# B&R Automation Studio project Y4_V3_1 (part 4)

#### SeamersCyclic.st - Cyclic code
```iecst
(********************************************************************
 * COPYRIGHT --
 ********************************************************************
 * Program: Seamers
 * File: SeamersCyclic.st
 * Author: nicke
 ********************************************************************
 * Implementation of program Seamers
 ********************************************************************)

PROGRAM _CYCLIC

//	Seamers.ESClear := Control.ESClear ;
//	Seamers.ControlIN := Control.Achieved1 ;
//	Seamers.Detension := Sol20DT1.Auto ;
//	Seamers.BeltsPT := PresetSys.Belt ;
//	Seamers.VacPT := PresetSys.Vac ;
//	Seamers.VacsStopPT := PresetSys.VacsStop ;
//	Seamers.PumpPT := PresetSys.Water ;
//	Seamers.Trips[1] := MS1Belt1.Trip ;
//	Seamers.Trips[2] := MS2Belt2.Trip ;
//	Seamers.Trips[4] := MS9Vac1.Trip ;
//	Seamers.Trips[7] := MS3Belt3.Trip ;
//	Seamers.Trips[8] := MS4Belt4.Trip ;
//	Seamers.Trips[10] := MS10Vac2.Trip ;
//	Seamers.Trips[13] := MS5Belt5.Trip ;
//	Seamers.Trips[14] := MS6Belt6.Trip ;
//	Seamers.Trips[16] := MS11Vac3.Trip ;
//	Seamers.Trips[19] := MS7Belt7.Trip ;
//	Seamers.Trips[20] := MS8Belt8.Trip ;
//	Seamers.Trips[22] := MS12Vac4.Trip ;
//	Seamers.Float[1] := S64Float.In ;
//	Seamers.Float[2] := S65Float.In ;
//	Seamers ();
//	MS1Belt1.Auto := Seamers.BeltOUT[1] ;
//	MS2Belt2.Auto := Seamers.BeltOUT[2] ;
//	MS3Belt3.Auto := Seamers.BeltOUT[3] ;
//	MS4Belt4.Auto := Seamers.BeltOUT[4] ;
//	MS5Belt5.Auto := Seamers.BeltOUT[5] ;
//	MS6Belt6.Auto := Seamers.BeltOUT[6] ;
//	MS7Belt7.Auto := Seamers.BeltOUT[7] ;
//	MS8Belt8.Auto := Seamers.BeltOUT[8] ;
//	MS9Vac1.Auto := Seamers.VacOUT[1] ;
//	MS11Vac3.Auto := Seamers.VacOUT[2] ;
//	MS10Vac2.Auto := Seamers.VacOUT[3] ;
//	MS12Vac4.Auto := Seamers.VacOUT[4] ;
//	Sol19Pump.Auto := Seamers.PumpOUT[0] ;
//	MS13Water1.Auto := Seamers.PumpOUT[1] ;
//	MS14Water2.Auto := Seamers.PumpOUT[2] ;
//	Seamers.StartAllDisp ;

	(*
	Intercept Interval delay TO be cumulative value OF time that spray nozzles are on (when seaming)
	Use counter FOR scans instead OF TON delay.
	CASE statement OF count FOR interval. Keep TON FOR Open delay.

	Timer in system, as glass is coming round, and times out, pauses line, shuts off the water pump AND vacuum pump FOR a few seconds FOR the bladder TO drain.
	Interval delay between drains.
	*)
	SeamersII.Control.Achieved := Control.Achieved1;
	SeamersII.Control.ESClear := Control.ESClear;
	SeamersII.Detension := Sol20DT1.Auto;
	SeamersII.PresetSys.Belt := PresetSys.Belt;
	SeamersII.PresetSys.Vac := PresetSys.Vac;
	SeamersII.PresetSys.VacsStop := PresetSys.VacsStop;
	SeamersII.PresetSys.Water := PresetSys.Water;
	SeamersII.Trips := SysTemp.Alarms;
	SeamersII.Float[1] := S64Float.In;
	SeamersII.SeekBlock[1] := Ax1.Block;
	SeamersII.SeekBlock[2] := Ax2.Block;
	SeamersII.InterceptInterval := InterceptPT.IntervalPT;
	SeamersII.InterceptOpen := InterceptPT.OpenPT;
	SeamersII ();
	MS1Belt1.Auto := SeamersII.BeltOUT[1];
	MS2Belt2.Auto := SeamersII.BeltOUT[2];
	MS3Belt3.Auto := SeamersII.BeltOUT[3];
	MS4Belt4.Auto := SeamersII.BeltOUT[4];
	MS5Belt5.Auto := SeamersII.BeltOUT[5];
	MS6Belt6.Auto := SeamersII.BeltOUT[6];
	MS7Belt7.Auto := SeamersII.BeltOUT[7];
	MS8Belt8.Auto := SeamersII.BeltOUT[8];
	MS9Vac1.Auto := SeamersII.VacOUT[1];
	MS10Vac2.Auto := SeamersII.VacOUT[2];
	MS11Vac3.Auto := SeamersII.VacOUT[3];
	MS12Vac4.Auto := SeamersII.VacOUT[4];
	Sol19Pump.Auto := SeamersII.ValveOUT[2];
	MS13Water1.Auto := SeamersII.PumpOUT[1];

	// NEW SPRAY NOZZLE CONTROL BASED ON U21
	// TURN ON SECOND PUMP WHEN FIRST VACUUM PUMP IS ON
	MS14Water2.Auto := (MS9Vac1.Auto) OR(MS11Vac3.Auto);
	IF(SeamersII.TransportMode)THEN
		MS14Water2.Auto := FALSE;
	END_IF
	IF NOT(S65Float.In)THEN
		MS14Water2.Auto := FALSE;
	END_IF

	// DON'T USE PRE TRACKING. TURNS SPRAY OFF
//	Spray1.PreTracking := 0; //CHANGE IF PRETRACKING REQUIRED
	Spray1.Track[0] := Track004.Active;
	Spray1.Track[1] := Track005.Active AND NOT(Tracking00.Blocked);
	Spray1.Track[2] := Track101.Active;
	Spray1.Track[3] := Track104.Active;
	Spray1.VacuumStopDelay := PresetSys.VacsStop;
	Spray1.NozzlePerm := NozzlePerm;
	Spray1.Vacuum := MS10Vac2.Auto;
	Spray1.AutoStart := SeamersII.AutoStart[1];
	Spray1.Control := Control.Achieved1;
	Spray1.TransportMode := SeamersII.TransportMode;
	Spray1 ();
	Sol37Spray.Auto := Spray1.Spray;// UNCOMMENT AFTER TESTING

	//ADD CONDITIONS TO RESET SEQUENCE FROM ALL CASES.

	// DON'T USE PRE TRACKING. TURNS SPRAY OFF
	Spray2.Track[0] := Track114.Active;
	Spray2.Track[1] := Track115.Active AND NOT(Tracking11.Blocked);
	Spray2.Track[2] := Track201.Active;
	Spray2.Track[3] := Track204.Active;
	Spray2.VacuumStopDelay := PresetSys.VacsStop;
	Spray2.NozzlePerm := NozzlePerm;
	Spray2.Vacuum := MS10Vac2.Auto;
	Spray2.AutoStart := SeamersII.AutoStart[1];
	Spray2.Control := Control.Achieved1;
	Spray2.TransportMode := SeamersII.TransportMode;
	Spray2 ();
	Sol47Spray.Auto := Spray2.Spray; //UNCOMMENT AFTER TESTING

	//RECIRCULATION VALVE - OPERATE WHEN BOTH SPRAY NOZZLE SOLENOIDS ARE OFF
	Sol53Recirc.Auto := FALSE;
	IF(Spray1.Nozzle.Seq >= NC_CleanDone) AND(Spray2.Nozzle.Seq >= NC_CleanDone)THEN
		IF(Sol37Spray.Auto = FALSE) AND(Sol47Spray.Auto = FALSE)THEN
			Sol53Recirc.Auto := TRUE;
		END_IF
	END_IF

END_PROGRAM
```

### Program Logical/System/SensorInput (IEC) - Anti blip for sensor inputs

#### SensorInputCyclic.st - Cyclic code
```iecst
//*******************************************************************
// * COPYRIGHT --
// ********************************************************************
// * Program: SensorInput
// * File: SensorInputCyclic.st
// * Author: nicke
// ********************************************************************
// * Implementation of program SensorInput
// *******************************************************************//

PROGRAM _CYCLIC

	Speeds.SpeedBatch:= LIMIT(1, Speeds.SpeedBatch, 60);
	Speeds.SpeedCntr:= LIMIT(1, Speeds.SpeedCntr, 60);
	Speeds.SpeedEntry:= LIMIT(1, Speeds.SpeedEntry, 60);
	Speeds.SpeedExit:= LIMIT(1, Speeds.SpeedExit, 60);
	Speeds.SpeedLaser:= LIMIT(1, Speeds.SpeedLaser, 60);
	Speeds.SpeedMax:= LIMIT(1, Speeds.SpeedMax, 60);
	Speeds.SpeedSeam:= LIMIT(1, Speeds.SpeedSeam, 60);
	Speeds.SpeedSlow:= LIMIT(1, Speeds.SpeedSlow, 60);
	Speeds.SpeedTrans:= LIMIT(1, Speeds.SpeedTrans, 60);
	Speeds.SpeedWash:= LIMIT(1, Speeds.SpeedWash, 60);
	Speeds.SpeedSeamSlow:= LIMIT(1, Speeds.SpeedSeamSlow, 60);

	//FILTER SENSOR 1 INPUT TO ELIMINATE FALSE READINGS
	//FB INPUTS
	Sensor1.SensorIN := S1Photo.In ;
	Sensor1.SpeedON := Speeds.SpeedTrans ;
	Sensor1.SpeedOFF := Speeds.SpeedSeam ;
	//CALL FB
	Sensor1 ();
	//FB OUTPUT
	S1Photo.Int := Sensor1.SensorOUT ;

	//FILTER SENSOR 2 INPUT TO ELIMINATE FALSE READINGS
	//FB INPUTS
	Sensor2.SensorIN := S2Photo.In ;
	Sensor2.SpeedON := Speeds.SpeedSlow ;
	Sensor2.SpeedOFF := Speeds.SpeedSeam ;
	//CALL FB
	Sensor2 ();
	//FB OUTPUT
	S2Photo.Int := Sensor2.SensorOUT ;

	//FILTER SENSOR 3 INPUT TO ELIMINATE FALSE READINGS
	//FB INPUTS
	Sensor3.SensorIN := S3Photo.In ;
	Sensor3.SpeedON := Speeds.SpeedSeam ;
	Sensor3.SpeedOFF := Speeds.SpeedSeam ;
	//CALL FB
	Sensor3 ();
	//FB OUTPUT
	S3Photo.Int := Sensor3.SensorOUT ;

	//FILTER SENSOR 4 INPUT TO ELIMINATE FALSE READINGS
	//FB INPUTS
	Sensor4.SensorIN := S4Photo.In ;
	Sensor4.SpeedON := Speeds.SpeedSeam ;
	Sensor4.SpeedOFF := Speeds.SpeedSeam ;
	//CALL FB
	Sensor4 ();
	//FB OUTPUT
	S4Photo.Int := Sensor4.SensorOUT ;

	//FILTER SENSOR 5 INPUT TO ELIMINATE FALSE READINGS
	//FB INPUTS
	Sensor5.SensorIN := S5Photo.In ;
	Sensor5.SpeedON := Speeds.SpeedTrans ;
	Sensor5.SpeedOFF := Speeds.SpeedSeam ;
	//CALL FB
	Sensor5 ();
	//FB OUTPUT
	S5Photo.Int := Sensor5.SensorOUT ;

	//FILTER SENSOR 6 INPUT TO ELIMINATE FALSE READINGS
	//FB INPUTS
	Sensor6.SensorIN := S6Photo.In ;
	Sensor6.SpeedON := Speeds.SpeedSlow ;
	Sensor6.SpeedOFF := Speeds.SpeedSeam ;
	//CALL FB
	Sensor6 ();
	//FB OUTPUT
	S6Photo.Int := Sensor6.SensorOUT ;

	//FILTER SENSOR 7 INPUT TO ELIMINATE FALSE READINGS
	//FB INPUTS
	Sensor7.SensorIN := S7Photo.In ;
	Sensor7.SpeedON := Speeds.SpeedSeam ;
	Sensor7.SpeedOFF := Speeds.SpeedSeam ;
	//CALL FB
	Sensor7 ();
	//FB OUTPUT
	S7Photo.Int := Sensor7.SensorOUT ;

	//FILTER SENSOR 8 INPUT TO ELIMINATE FALSE READINGS
	//FB INPUTS
	Sensor8.SensorIN := S8Photo.In ;
	Sensor8.SpeedON := Speeds.SpeedSeam ;
	Sensor8.SpeedOFF := Speeds.SpeedSeam ;
	//CALL FB
	Sensor8 ();
	//FB OUTPUT
	S8Photo.Int := Sensor8.SensorOUT ;

	//FILTER SENSOR 9 INPUT TO ELIMINATE FALSE READINGS
	//FB INPUTS
	Sensor9.SensorIN := S9Photo.In ;
	Sensor9.SpeedON := Speeds.SpeedSeam ;
	Sensor9.SpeedOFF := Speeds.SpeedSeam ;
	//CALL FB
	Sensor9 ();
	//FB OUTPUT
	S9Photo.Int := Sensor9.SensorOUT ;

	//FILTER SENSOR 12 INPUT TO ELIMINATE FALSE READINGS
	//FB INPUTS
	Sensor12.SensorIN := S12Photo.In ;
	Sensor12.SpeedON := Speeds.SpeedSeam ;
	Sensor12.SpeedOFF := Speeds.SpeedTrans ;
	//CALL FB
	Sensor12 ();
	//FB OUTPUT
	S12Photo.Int := Sensor12.SensorOUT ;

	//FILTER SENSOR 13 INPUT TO ELIMINATE FALSE READINGS
	//FB INPUTS
	Sensor13.SensorIN := S13Photo.In ;
	Sensor13.SpeedON := Speeds.SpeedExit ;
	Sensor13.SpeedOFF := Speeds.SpeedExit ;
	//CALL FB
	Sensor13 ();
	//FB OUTPUT
	S13Photo.Int := Sensor13.SensorOUT ;

	//FILTER SENSOR 14 INPUT TO ELIMINATE FALSE READINGS
	//FB INPUTS
	Sensor14.SensorIN := S14Photo.In ;
	Sensor14.SpeedON := Speeds.SpeedExit ;
	Sensor14.SpeedOFF := Speeds.SpeedExit ;
	//CALL FB
	Sensor14 ();
	//FB OUTPUT
	S14Photo.Int := Sensor14.SensorOUT ;

	//FILTER SENSOR 15 INPUT TO ELIMINATE FALSE READINGS
	//FB INPUTS
	Sensor15.SensorIN := S15Photo.In ;
	Sensor15.SpeedON := Speeds.SpeedExit ;
	Sensor15.SpeedOFF := Speeds.SpeedExit ;
	//CALL FB
	Sensor15 ();
	//FB OUTPUT
	S15Photo.Int := Sensor15.SensorOUT ;

	//FILTER SENSOR 16 INPUT TO ELIMINATE FALSE READINGS
	//FB INPUTS
	Sensor16.SensorIN := S16Photo.In ;
	Sensor16.SpeedON := Speeds.SpeedExit ;
	Sensor16.SpeedOFF := Speeds.SpeedExit ;
	//CALL FB
	Sensor16 ();
	//FB OUTPUT
	S16Photo.Int := Sensor16.SensorOUT ;

	//FILTER SENSOR 17 INPUT TO ELIMINATE FALSE READINGS
	//FB INPUTS
	Sensor17.SensorIN := S17Photo.In ;
	Sensor17.SpeedON := Speeds.SpeedExit ;
	Sensor17.SpeedOFF := Speeds.SpeedExit ;
	//CALL FB
	Sensor17 ();
	//FB OUTPUT
	S17Photo.Int := Sensor17.SensorOUT ;

	//FILTER SENSOR 18 INPUT TO ELIMINATE FALSE READINGS
	//FB INPUTS
	Sensor18.SensorIN := S18Photo.In ;
	Sensor18.SpeedON := Speeds.SpeedCntr ;
	Sensor18.SpeedOFF := Speeds.SpeedCntr ;
	//CALL FB
	Sensor18 ();
	//FB OUTPUT
	S18Photo.Int := Sensor18.SensorOUT ;

	//FILTER SENSOR 19 INPUT TO ELIMINATE FALSE READINGS
	//FB INPUTS
	Sensor19.SensorIN := S19Photo.In ;
	Sensor19.SpeedON := Speeds.SpeedBatch ;
	Sensor19.SpeedOFF := Speeds.SpeedBatch ;
	//CALL FB
	Sensor19 ();
	//FB OUTPUT
	S19Photo.Int := Sensor19.SensorOUT ;

	//FILTER SENSOR 20 INPUT TO ELIMINATE FALSE READINGS
	//FB INPUTS
	Sensor20.SensorIN := S20Photo.In ;
	Sensor20.SpeedON := Speeds.SpeedBatch ;
	Sensor20.SpeedOFF := Speeds.SpeedBatch ;
	//CALL FB
	Sensor20 ();
	//FB OUTPUT
	S20Photo.Int := Sensor20.SensorOUT ;

	//FILTER SENSOR 21 INPUT TO ELIMINATE FALSE READINGS
	//FB INPUTS
	Sensor21.SensorIN := S21Photo.In ;
	Sensor21.SpeedON := Speeds.SpeedBatch ;
	Sensor21.SpeedOFF := Speeds.SpeedWash ;
	//CALL FB
	Sensor21 ();
	//FB OUTPUT
	S21Photo.Int := Sensor21.SensorOUT ;

END_PROGRAM
```

### Program Logical/System/Process (IEC) - Operation information

#### ProcessCyclic.st - Cyclic code
```iecst
(********************************************************************
 * COPYRIGHT -ASHTON INDUSTRIAL 2016-
 ********************************************************************
 * Program: Process
 * Author: NE
 ********************************************************************)

PROGRAM _CYCLIC

	//CALCULATION FOR MACHINE RUN TIME. DISPLAYED IN YY:DD:HH:MM
	//FB INPUTS
	RunTime1.On := Control.Achieved1 ;
	RunTime1.TotReset := Reset.Total ;
	RunTime1.ShftReset := Reset.Time ;
	RunTime1.TotMinIn := Data.TotalMins ;
	RunTime1.TotHrIn := Data.TotalHrs ;
	RunTime1.TotDayIn := Data.TotalDays ;
	RunTime1.TotYrIn := Data.TotalYrs ;
	RunTime1.ShftMinIn := Data.ShiftMins ;
	RunTime1.ShftHrIn := Data.ShiftHrs ;
	RunTime1.ShftDayIn := Data.ShiftDays ;
	RunTime1.ShftYrIn := Data.ShiftYrs ;
	//CALL FB
	RunTime1();
	//FB OUTPUTS
	Data.TotalMins := RunTime1.TotMin ;
	Data.TotalHrs := RunTime1.TotHr ;
	Data.TotalDays := RunTime1.TotDay ;
	Data.TotalYrs := RunTime1.TotYr ;
	Data.ShiftMins := RunTime1.ShftMin ;
	Data.ShiftHrs := RunTime1.ShftHr ;
	Data.ShiftDays := RunTime1.ShftDay ;
	Data.ShiftYrs := RunTime1.ShftYr ;

	//CALCULATE BELT GRIND TIMES FOR WIDTH. DISPLAYED IN DD:HH:MM:SS
	//TRACKING BIT TRIGGER FOR CALCULATION
	GrindFB1.On := FALSE ;
	GrindFB1M.On := FALSE ;
	IF EDGEPOS(Seaming.Stop2) THEN
		GrindFB1.On := TRUE ;
		GrindFB1M.On := TRUE ;
	END_IF

	//FB INPUTS
	GrindFB1.TotReset := Reset.Total ;
	GrindFB1.ShftReset := Reset.Grind ;
	GrindFB1M.ShftReset := MeterageReset1.Reset ;
	IF (ProcessMode.In) THEN
		GrindFB1.Speed := Speeds.SpeedSeamSlow;
	ELSE
		GrindFB1.Speed := Speeds.SpeedSeam ;
	END_IF
	GrindFB1.Measured := Ax2.Measure/10 ;
	GrindFB1.TotMSIn := Grind1.TotalMs ;
	GrindFB1.TotSecIn := Grind1.TotalSec ;
	GrindFB1.TotMinIn := Grind1.TotalMin ;
	GrindFB1.TotHrIn := Grind1.TotalHr ;
	GrindFB1.TotDayIn := Grind1.TotalDay ;
	GrindFB1.ShftMSIn := Grind1.ShiftMs ;
	GrindFB1.ShftSecIn := Grind1.ShiftSec ;
	GrindFB1.ShftMinIn := Grind1.ShiftMin ;
	GrindFB1.ShftHrIn := Grind1.ShiftHr ;
	GrindFB1.ShftDayIn := Grind1.ShiftDay ;
	GrindFB1.TotMtrs1In := Grind1.TotalMLow ;
	GrindFB1.TotMtrs2In := Grind1.TotalMUpp ;
	GrindFB1.TotFt1In := Grind1.TotalFtLow ;
	GrindFB1.TotFt2In := Grind1.TotalFtUpp ;
	GrindFB1M.Measured := GrindFB1.Measured;
 	GrindFB1M.ShftMtrs1In := Grind1.ShiftMLow ;
	GrindFB1M.ShftMtrs2In := Grind1.ShiftMUpp ;
	GrindFB1.ShftFt1In := Grind1.ShiftFtLow ;
	GrindFB1.ShftFt2In := Grind1.ShiftFtUpp ;
	//CALL FB
	GrindFB1();
	GrindFB1M ();
	//FB OUTPUTS
	Grind1.TotalMs := GrindFB1.TotMS ;
	Grind1.TotalSec := GrindFB1.TotSec ;
	Grind1.TotalMin := GrindFB1.TotMin ;
	Grind1.TotalHr := GrindFB1.TotHr ;
	Grind1.TotalDay := GrindFB1.TotDay ;
	Grind1.ShiftMs := GrindFB1.ShftMS ;
	Grind1.ShiftSec := GrindFB1.ShftSec ;
	Grind1.ShiftMin := GrindFB1.ShftMin ;
	Grind1.ShiftHr := GrindFB1.ShftHr ;
	Grind1.ShiftDay := GrindFB1.ShftDay ;
	Grind1.TotalMLow := GrindFB1.TotMtrs1 ;
	Grind1.TotalMUpp := GrindFB1.TotMtrs2 ;
	Grind1.TotalFtLow := GrindFB1.TotFt1 ;
	Grind1.TotalFtUpp := GrindFB1.TotFt2 ;
	Grind1.ShiftMLow := GrindFB1M.ShftMtrs1 ;
	Grind1.ShiftMUpp := GrindFB1M.ShftMtrs2 ;
	Grind1.ShiftFtLow := GrindFB1.ShftFt1 ;
	Grind1.ShiftFtUpp := GrindFB1.ShftFt2 ;

	//CALCULATE BELT GRIND TIMES FOR LENGTH. DISPLAYED IN DD:HH:MM:SS
	//TRACKING BIT TRIGGER FOR CALCULATION
	GrindFB2.On := FALSE ;
	GrindFB2M.On := FALSE ;
	IF EDGEPOS(Seaming.Stop2) THEN
		GrindFB2.On := TRUE ;
		GrindFB2M.On := TRUE ;
	END_IF
	//FB INPUTS
	GrindFB2.TotReset := Reset.Total ;
	GrindFB2.ShftReset := Reset.Grind ;
	GrindFB2M.ShftReset := MeterageReset2.Reset ;
	IF (ProcessMode.In) THEN
		GrindFB2.Speed := Speeds.SpeedSeamSlow;
	ELSE
		GrindFB2.Speed := Speeds.SpeedSeam ;
	END_IF
	GrindFB2.Measured := Tracking20.Length ;
	GrindFB2.TotMSIn := Grind2.TotalMs ;
	GrindFB2.TotSecIn := Grind2.TotalSec ;
	GrindFB2.TotMinIn := Grind2.TotalMin ;
	GrindFB2.TotHrIn := Grind2.TotalHr ;
	GrindFB2.TotDayIn := Grind2.TotalDay ;
	GrindFB2.ShftMSIn := Grind2.ShiftMs ;
	GrindFB2.ShftSecIn := Grind2.ShiftSec ;
	GrindFB2.ShftMinIn := Grind2.ShiftMin ;
	GrindFB2.ShftHrIn := Grind2.ShiftHr ;
	GrindFB2.ShftDayIn := Grind2.ShiftDay ;
	GrindFB2.TotMtrs1In := Grind2.TotalMLow ;
	GrindFB2.TotMtrs2In := Grind2.TotalMUpp ;
	GrindFB2.TotFt1In := Grind2.TotalFtLow ;
	GrindFB2.TotFt2In := Grind2.TotalFtUpp ;
	GrindFB2M.Measured := GrindFB2.Measured;
	GrindFB2M.ShftMtrs1In := Grind2.ShiftMLow ;
	GrindFB2M.ShftMtrs2In := Grind2.ShiftMUpp ;
	GrindFB2.ShftFt1In := Grind2.ShiftFtLow ;
	GrindFB2.ShftFt2In := Grind2.ShiftFtUpp ;
	//CALL FB
	GrindFB2();
	GrindFB2M();
	//FB OUTPUTS
	Grind2.TotalMs := GrindFB2.TotMS ;
	Grind2.TotalSec := GrindFB2.TotSec ;
	Grind2.TotalMin := GrindFB2.TotMin ;
	Grind2.TotalHr := GrindFB2.TotHr ;
	Grind2.TotalDay := GrindFB2.TotDay ;
	Grind2.ShiftMs := GrindFB2.ShftMS ;
	Grind2.ShiftSec := GrindFB2.ShftSec ;
	Grind2.ShiftMin := GrindFB2.ShftMin ;
	Grind2.ShiftHr := GrindFB2.ShftHr ;
	Grind2.ShiftDay := GrindFB2.ShftDay ;
	Grind2.TotalMLow := GrindFB2.TotMtrs1 ;
	Grind2.TotalMUpp := GrindFB2.TotMtrs2 ;
	Grind2.TotalFtLow := GrindFB2.TotFt1 ;
	Grind2.TotalFtUpp := GrindFB2.TotFt2 ;
	Grind2.ShiftMLow := GrindFB2M.ShftMtrs1 ;
	Grind2.ShiftMUpp := GrindFB2M.ShftMtrs2 ;
	Grind2.ShiftFtLow := GrindFB2.ShftFt1 ;
	Grind2.ShiftFtUpp := GrindFB2.ShftFt2 ;

	//COMPARE SHIFT METERS AND SET WARNING WHEN GREATER
	Meterage1 := FB_HIDE;
	Meterage2 := FB_HIDE;
	Warn.Timeout[30] := FALSE;
	Warn.Timeout[31] := FALSE;
	IF (Grind1.ShiftMLow > TrackDelayPT.PTTrack913) THEN
		Meterage1 := FB_SHOW;
		Warn.Timeout[30] := TRUE;
	END_IF
	IF (Grind2.ShiftMLow > TrackDelayPT.PTTrack922) THEN
		Meterage2 := FB_SHOW;
		Warn.Timeout[31] := TRUE;
	END_IF

	//PIECE COUNT
	IF EDGENEG(Seaming.Stop2) AND(Control.Achieved1) THEN
		Data.TotalPiece := Data.TotalPiece + 1 ;
		Data.ShiftPiece := Data.ShiftPiece + 1 ;
	END_IF

	//RESET TOTAL
	IF (Reset.Total) THEN
		Data.TotalPiece := 0 ;
	END_IF

	//RESET SHIFT TOTAL
	IF (Reset.Count) THEN
		Data.ShiftPiece := 0 ;
	END_IF

END_PROGRAM
```

### Program Logical/System/IO (IEC) - IO addressing

#### IOCyclic.st - Cyclic code
```iecst
(********************************************************************
 * COPYRIGHT --
 ********************************************************************
 * Program: IO
 * File: IOCyclic.st
 * Author: nicke
 ********************************************************************
 * Implementation of program IO
 ********************************************************************)

PROGRAM _CYCLIC

	IF NOT(Simulation.On) THEN  //DISABLE WHEN SIMULATION RUNNING
		//MAP X2X ST02 TO VARIABLES
		Control.Start := X2X02.P1 ;
		Control.Stop := X2X02.P2 ;
		Control.EStop1 := X2X02.P3 ;
		X2X02.P4 ;
		MS1Belt1.Trip := X2X02.P5 ;
		MS2Belt2.Trip := X2X02.P6 ;
		MS3Belt3.Trip := X2X02.P7 ;
		MS4Belt4.Trip := X2X02.P8 ;
		MS5Belt5.Trip := X2X02.P9 ;
		MS6Belt6.Trip := X2X02.P10 ;
		MS7Belt7.Trip := X2X02.P11 ;
		MS8Belt8.Trip := X2X02.P12 ;
		//MAP X2X ST03 TO VARIABLES
		MS9Vac1.Trip := X2X03.P1 ;
		MS10Vac2.Trip := X2X03.P2 ;
		MS11Vac3.Trip := X2X03.P3 ;
		MS12Vac4.Trip := X2X03.P4 ;
		MS13Water1.Trip := X2X03.P5 ;
		MS14Water2.Trip := X2X03.P6 ;
		X2X03.P7 ;
		X2X03.P8 ;
		X2X03.P9 ;
		X2X03.P10 ;
		X2X03.P11 ;
		ClearBatch.In := X2X03.P12 ;
		//MAP X2X ST04 TO VARIABLES
		X2X04.P1 := Control.Buzzer ;
		X2X04.P2 := Control.OnLmp1 ;
		X2X04.P3 ;
		X2X04.P4 ;
		X2X04.P5 ;
		X2X04.P6 ;
		X2X04.P7 ;
		X2X04.P8 ;
		X2X04.P9 ;
		X2X04.P10 ;
		X2X04.P11 := SEL(Control.Auto,Sol24DG1B.Test,Sol24DG1B.Auto) ;
		X2X04.P12 := Filstar.Out ;
		//MAP X2X ST08 TO VARIABLES
		X2X08.P1 := SEL(Control.Auto,MS1Belt1.Test,MS1Belt1.Auto) ;
		X2X08.P2 := SEL(Control.Auto,MS2Belt2.Test,MS2Belt2.Auto) ;
		X2X08.P3 := SEL(Control.Auto,MS3Belt3.Test,MS3Belt3.Auto) ;
		X2X08.P4 := SEL(Control.Auto,MS4Belt4.Test,MS4Belt4.Auto) ;
		X2X08.P5 := SEL(Control.Auto,MS5Belt5.Test,MS5Belt5.Auto) ;
		X2X08.P6 := SEL(Control.Auto,MS6Belt6.Test,MS6Belt6.Auto) ;
		X2X08.P7 := SEL(Control.Auto,MS7Belt7.Test,MS7Belt7.Auto) ;
		X2X08.P8 := SEL(Control.Auto,MS8Belt8.Test,MS8Belt8.Auto) ;
		X2X08.P9 := SEL(Control.Auto,MS9Vac1.Test,MS9Vac1.Auto) ;
		X2X08.P10 := SEL(Control.Auto,MS10Vac2.Test,MS10Vac2.Auto) ;
		X2X08.P11 := SEL(Control.Auto,MS11Vac3.Test,MS11Vac3.Auto) ;
		X2X08.P12 := SEL(Control.Auto,MS12Vac4.Test,MS12Vac4.Auto) ;
		X2X08.P13 := SEL(Control.Auto,MS13Water1.Test,MS13Water1.Auto) ;
		X2X08.P14 := SEL(Control.Auto,MS14Water2.Test,MS14Water2.Auto) ;
		X2X08.P15 ;
		X2X08.P16 ;
		//MAP X2X ST10 TO VARIABLES
		S45Foot.In := X2X10.P1 ;
		S1Photo.In := X2X10.P2 ;
		S2Photo.In := X2X10.P3 ;
		S56Lever.In := X2X10.P4 ;
		S30Reed.In := X2X10.P5 ;
		S31Reed.In := X2X10.P6 ;
		LaserBusy.In := X2X10.P7 ;
		X2X10.P8 := LaserFire.Auto ;
		S100Reed.In := X2X10.P9 ;
		X2X10.P10 := SEL(Control.Auto,Sol37Spray.Test,Sol37Spray.Auto) ;
		X2X10.P11 := SEL(Control.Auto,Sol2Blt2.Test,Sol2Blt2.Auto) ;
		X2X10.P12 := SEL(Control.Auto,Sol5Arm1.Test,Sol5Arm1.Auto) ;
		X2X10.P13 := SEL(Control.Auto,Sol6Arm2.Test,Sol6Arm2.Auto) ;
		X2X10.P14 := SEL(Control.Auto,Sol7Arm3.Test,Sol7Arm3.Auto) ;
		X2X10.P15 := SEL(Control.Auto,Sol8Arm4.Test,Sol8Arm4.Auto) ;
		X2X10.P16 := SEL(Control.Auto,Sol20DT1.Test,Sol20DT1.Auto) ;
		//MAP X2X ST11 TO VARIABLES
		S81Photo.In := X2X11.P1 ;
		S82Photo.In := X2X11.P2 ;
		S83Photo.In := X2X11.P3 ;
		S84Photo.In := X2X11.P4 ;
		X2X11.P5 := SEL(Control.Auto,Sol3Blt3.Test,Sol3Blt3.Auto) ;
		X2X11.P6 := SEL(Control.Auto,Sol4Blt4.Test,Sol4Blt4.Auto) ;
		X2X11.P7 := SEL(Control.Auto,Sol21DT2.Test,Sol21DT2.Auto) ;
		S3Photo.In := X2X11.P8 ;
		//MAP X2X ST12 TO VARIABLES
		Servo1POT.In := X2X12.P1 ;
		Servo1NOT.In := X2X12.P2 ;
		S80Origin.In := X2X12.P3 ;
		S101Reed.In := X2X12.P4 ;
		S104Reed.In := X2X12.P5 ;
		S105Reed.In := X2X12.P6 ;
		S106Reed.In := X2X12.P7 ;
		S107Reed.In := X2X12.P8 ;
		S108Reed.In := X2X12.P9 ;
		S109Reed.In := X2X12.P10 ;
		S110Reed.In := X2X12.P11 ;
		S111Reed.In := X2X12.P12 ;
		S112Reed.In := X2X12.P13 ;
		S113Reed.In := X2X12.P14 ;
		S114Reed.In := X2X12.P15 ;
		S115Reed.In := X2X12.P16 ;
		//MAP X2X ST13 TO VARIABLES
		S4Photo.In := X2X13.P1 ;
		S5Photo.In := X2X13.P2 ;
		S6Photo.In := X2X13.P3 ;
		S9Photo.In := X2X13.P4 ;
		S32Reed.In := X2X13.P5 ;
		S33Reed.In := X2X13.P6 ;
		S50Reed.In := X2X13.P7 ;
		S102Reed.In := X2X13.P8 ;
		S103Reed.In := X2X13.P9 ;
		X2X13.P10 := SEL(Control.Auto,Sol30Pal1.Test,Sol30Pal1.Auto) ;
		X2X13.P11 := SEL(Control.Auto,Sol31Pal2.Test,Sol31Pal2.Auto) ;
		X2X13.P12 := SEL(Control.Auto,Sol32Pal3.Test,Sol32Pal3.Auto) ;
		X2X13.P13 := SEL(Control.Auto,Sol33Pal4.Test,Sol33Pal4.Auto) ;
		X2X13.P14 := SEL(Control.Auto,Sol24DG1.Test,Sol24DG1.Auto) ;
		X2X13.P15 := Sol35Laser.Auto ;
		X2X13.P16 := SEL(Control.Auto,Sol19Pump.Test,Sol19Pump.Auto) ;
		//MAP X2X ST14 TO VARIABLES
		X2X14.P1 := SEL(Control.Auto,Sol47Spray.Test,Sol47Spray.Auto) ;
		X2X14.P2 := SEL(Control.Auto,Sol53Recirc.Test,Sol53Recirc.Auto) ;
		X2X14.P3 := SEL(Control.Auto,Sol14Arm6.Test,Sol14Arm6.Auto) ;
		X2X14.P4 := SEL(Control.Auto,Sol15Arm7.Test,Sol15Arm7.Auto) ;
		X2X14.P5 := SEL(Control.Auto,Sol22DT3.Test,Sol22DT3.Auto) ;
		S7Photo.In := X2X14.P6 ;
		S64Float.In := X2X14.P7 ;
		S65Float.In := X2X14.P8 ;
		//MAP X2X ST15 TO VARIABLES
		Servo2POT.In := X2X15.P1 ;
		Servo2NOT.In := X2X15.P2 ;
		S90Origin.In := X2X15.P3 ;
		S12Photo.In := X2X15.P4 ;
		S13Photo.In := X2X15.P5 ;
		S34Reed.In := X2X15.P6 ;
		S35Reed.In := X2X15.P7 ;
		X2X15.P8 ;
		S120Reed.In := X2X15.P9 ;
		S121Reed.In := X2X15.P10 ;
		S122Reed.In := X2X15.P11 ;
		S123Reed.In := X2X15.P12 ;
		S124Reed.In := X2X15.P13 ;
		S125Reed.In := X2X15.P14 ;
		S126Reed.In := X2X15.P15 ;
		S127Reed.In := X2X15.P16 ;
		//MAP X2X ST16 TO VARIABLES
		S91Photo.In := X2X16.P1 ;
		S92Photo.In := X2X16.P2 ;
		S93Photo.In := X2X16.P3 ;
		S94Photo.In := X2X16.P4 ;
		X2X16.P5 := SEL(Control.Auto,Sol12Blt7.Test,Sol12Blt7.Auto) ;
		X2X16.P6 := SEL(Control.Auto,Sol13Blt8.Test,Sol13Blt8.Auto) ;
		X2X16.P7 := SEL(Control.Auto,Sol23DT4.Test,Sol23DT4.Auto) ;
		S8Photo.In := X2X16.P8 ;
		X2X16.P9 := SEL(Control.Auto,Sol40Datum.Test,Sol40Datum.Auto) ;
		X2X16.P10 ;
		X2X16.P11 ;
		X2X16.P12 ;
		S52Reed.In := X2X16.P13 ;
		S53Reed.In := X2X16.P14 ;
		X2X16.P15 ;
		X2X16.P16 ;
		//MAP X2X ST17 TO VARIABLES
		S14Photo.In := X2X17.P1 ;
		S15Photo.In := X2X17.P2 ;
		S16Photo.In := X2X17.P3 ;
		S17Photo.In := X2X17.P4 ;
		S18Photo.In := X2X17.P5 ;
		S36Reed.In := X2X17.P6 ;
		S37Reed.In := X2X17.P7 ;
		S57Lever.In := X2X17.P8 ;
		//MAP X2X ST18 TO VARIABLES
		S19Photo.In := X2X18.P1 ;
		X2X18.P2 ;
		X2X18.P3 ;
		X2X18.P4 ;
		S21Photo.In := X2X18.P5 ;
		X2X18.P6 ;
		S55Lever.In := X2X18.P7 ;
		WashRun.In := X2X18.P8 ;
		FurnReady.In := X2X18.P9 ;
		X2X18.P10 := WashStop.Auto ;
		X2X18.P11 := BatchAtExit.Auto ;
		S48Foot.In := X2X18.P12 ;
		S66PB.In := X2X18.P13 ;
		S58Lever.In := X2X18.P14 ;
		S20Photo.In := X2X18.P15 ;
		X2X18.P16 ; //INPUT CAN BE USED FOR BUTTON OR FOOTPEDAL TO BRING UP NEXT SCREEN ON BATCHING DISPLAY.
		//MAP X2X ST20 TO VARIABLES
		AGVReady.In := X2X20.P1;
		AGVInPosition.In := X2X20.P2;
		AGVReceiving.In := X2X20.P3;
		X2X20.P4;
		X2X20.P5;
		X2X20.P6;
		X2X20.P7;
		X2X20.P8;
		X2X20.P9;
		X2X20.P10;
		AGVAcknowledge.In := X2X20.P11;
		X2X20.P12;
		//MAP X2X ST21 TO VARIABLES
		X2X21.P1 := AGVRequired.Auto;
		X2X21.P2;
		X2X21.P3;
		X2X21.P4;
		X2X21.P5 := AGVReadyToSend.Auto;
		X2X21.P6;
		X2X21.P7 := AGVBatchClear.Auto;
		X2X21.P8 := SizeData.LengthMask;
		X2X21.P9 := SizeData.WidthMask;
		X2X21.P10 := AGVSending.Auto;
		X2X21.P11;
		X2X21.P12;
		//MAP X2X ST22 TO VARIABLES
		X2X22.P1 := SizeData.Sizes[0];
		X2X22.P2 := SizeData.Sizes[1];
		X2X22.P3 := SizeData.Sizes[2];
		X2X22.P4 := SizeData.Sizes[3];
		X2X22.P5 := SizeData.Sizes[4];
		X2X22.P6 := SizeData.Sizes[5];
		X2X22.P7 := SizeData.Sizes[6];
		X2X22.P8 := SizeData.Sizes[7];
		X2X22.P9 := SizeData.Sizes[8];
		X2X22.P10 := SizeData.Sizes[9];
		X2X22.P11 := SizeData.Sizes[10];
		X2X22.P12 := SizeData.Sizes[11];
	END_IF

	//RESET TEST BITS WHEN EXITING TEST SCREENS
	IF NOT(Control.Test) THEN
		Sol24DG1B.Test := FALSE ;
		MS1Belt1.Test := FALSE ;
		MS2Belt2.Test := FALSE ;
		MS3Belt3.Test := FALSE ;
		MS4Belt4.Test := FALSE ;
		MS5Belt5.Test := FALSE ;
		MS6Belt6.Test := FALSE ;
		MS7Belt7.Test := FALSE ;
		MS8Belt8.Test := FALSE ;
		MS9Vac1.Test := FALSE ;
		MS10Vac2.Test := FALSE ;
		MS11Vac3.Test := FALSE ;
		MS12Vac4.Test := FALSE ;
		MS13Water1.Test := FALSE ;
		MS14Water2.Test := FALSE ;
		Sol1Blt1.Test := FALSE ;
		Sol2Blt2.Test := FALSE ;
		Sol5Arm1.Test := FALSE ;
		Sol6Arm2.Test := FALSE ;
		Sol7Arm3.Test := FALSE ;
		Sol8Arm4.Test := FALSE ;
		Sol3Blt3.Test := FALSE ;
		Sol4Blt4.Test := FALSE ;
		Sol19Pump.Test := FALSE ;
		Sol21DT2.Test := FALSE ;
		Sol30Pal1.Test := FALSE ;
		Sol31Pal2.Test := FALSE ;
		Sol32Pal3.Test := FALSE ;
		Sol33Pal4.Test := FALSE ;
		Sol24DG1.Test := FALSE ;
		Sol10Blt5.Test := FALSE ;
		Sol11Blt6.Test := FALSE ;
		Sol14Arm6.Test := FALSE ;
		Sol15Arm7.Test := FALSE ;
		Sol12Blt7.Test := FALSE ;
		Sol13Blt8.Test := FALSE ;
		Sol23DT4.Test := FALSE ;
		Sol37Spray.Test := FALSE;
		Sol40Datum.Test := FALSE ;
		Sol47Spray.Test := FALSE;
		Sol53Recirc.Test := FALSE;
		CL1.Inv.Test := 0 ;
		CS1.Inv.Test := 0 ;
		CV1.Inv.Test := 0 ;
		CC1.Inv.Test := 0 ;
		CC2.Inv.Test := 0 ;
		CS2.Inv.Test := 0 ;
		CV2.Inv.Test := 0 ;
		CC3.Inv.Test := 0 ;
		CC4.Inv.Test := 0 ;
		CB1.Inv.Test := 0 ;
		CB2.Inv.Test := 0 ;
		CRB.Inv.Test := 0 ;
		CRE.Inv.Test := 0 ;
		CLB.Inv.Test := 0 ;
	END_IF

END_PROGRAM
```

### Program Logical/System/Filstar (IEC) - Filstar valve control

#### FilstarCyclic.st - Cyclic code
```iecst
(********************************************************************
 * COPYRIGHT --
 ********************************************************************
 * Program: Filstar
 * File: FilstarCyclic.st
 * Author: nicke
 * Created: February, 2012
 ********************************************************************
 * Implementation of program Filstar
 ********************************************************************)

PROGRAM _INIT

Filstar.Open.IN		:=	TRUE	;

END_PROGRAM

PROGRAM _CYCLIC

(*Delay for filstar valve open*)
Filstar.Open.PT	:=	PresetSys.Filstar[1]	;
Filstar.Open ();
(*Filstar valve control*)
Filstar.Out	:=	Filstar.Open.M	;

IF (Filstar.Open.Q) THEN
	Filstar.Open.IN		:=	FALSE	;
	Filstar.Interval.IN	:=	TRUE	;
END_IF
(*Delay for inteval between valve open*)
Filstar.Interval.PT	:=	PresetSys.Filstar[2]	;
Filstar.Interval ();

IF (Filstar.Interval.Q) THEN
	Filstar.Interval.IN	:= 	FALSE	;
	Filstar.Open.IN		:=	TRUE	;
END_IF

END_PROGRAM
```

### Program Logical/System/LineConfig (IEC) - IO Line Configuration

#### LineConfigCyclic.st - Cyclic code
```iecst
(********************************************************************
 * COPYRIGHT --
 ********************************************************************
 * Program: LineConfig
 * File: LineConfigCyclic.st
 * Author: nicke
 ********************************************************************)
PROGRAM _CYCLIC

	Perms.FLIPARMS1 := 4 ;
	Perms.FLIPARMS2 := 2 ;

	Perms.VersionText	:=	'S/W Version 3.1 02/26'	;

	// DeviceName used for mapping IO to ACOPOS
	Ax1.Node	:=	'SL1.IF1.ST1.IF1.ST12'	;	// Alter to suit each job
	Ax2.Node	:=	'SL1.IF1.ST1.IF1.ST15'	;	// Alter to suit each job

// Servo settings
	Ax1P.AbsMax	:=	40000				;	// Max Size of Axis 1
	Ax1P.AbsMin	:=	3000				;	// Min Size of Axis 1
	Ax2P.AbsMax	:=	25000				;	// Max Size of Axis 2
	Ax2P.AbsMin	:=	2000				;	// Min Size of Axis 2

	// Calculated limits for visu input
	Ax1.Max.Upp		:=	(Ax1P.AbsMax + 50)		;	// Maximum upper limit input
	Ax1.Max.Low		:=	(Ax1P.AbsMax/2)			;	// Maximum lower limit input
	Ax1.Max.UppF	:=	(Ax1P.AbsMax - 2000)	;	// Maximum feed upper limit input
	Ax1.Max.LowF	:=	(Ax1P.AbsMax - 2800)	;	// Maximum feed lower limit input
	Ax1.Max.UppO	:=	(Ax1P.AbsMax + 50)		;	// Maximum origin upper limit input
	Ax1.Max.LowO	:=	(Ax1P.AbsMax - 50)		;	// Maximum origin lower limit input
	Ax1.Min.Upp		:=	(Ax1P.AbsMax/2)			;	// Minimum upper limit input
	Ax1.Min.Low		:=	(Ax1P.AbsMin - 50)		;	// Minimum lower limit input
	Ax1.Min.UppF	:=	(Ax1P.AbsMin + 2000)	;	// Minimum feed upper limit input
	Ax1.Min.LowF	:=	(Ax1P.AbsMin + 3500)	;	// Minimum feed lower limit input
	Ax2.Max.Upp		:=	(Ax2P.AbsMax + 50)		;	// Maximum upper limit input
	Ax2.Max.Low		:=	(Ax2P.AbsMax/2)			;	// Maximum lower limit input
	Ax2.Max.UppF	:=	(Ax2P.AbsMax - 2000)	;	// Maximum feed upper limit input
	Ax2.Max.LowF	:=	(Ax2P.AbsMax - 2800)	;	// Maximum feed lower limit input
	Ax2.Max.UppO	:=	(Ax2P.AbsMax + 50)		;	// Maximum origin upper limit input
	Ax2.Max.LowO	:=	(Ax2P.AbsMax - 50)		;	// Maximum origin lower limit input
	Ax2.Min.Upp		:=	(Ax2P.AbsMax/2)			;	// Minimum upper limit input
	Ax2.Min.Low		:=	(Ax2P.AbsMin - 50)		;	// Minimum lower limit input
	Ax2.Min.UppF	:=	(Ax2P.AbsMin + 2000)	;	// Minimum feed upper limit input
	Ax2.Min.LowF	:=	(Ax2P.AbsMin + 3500)	;	// Minimum feed lower limit input

	//LIMIT INPUT VALUES FOR HMI
	RowPerm.Max		:=	LIMIT(150,RowPerm.Max,2489)	;//98"
	LoadPerm.Max	:=	LIMIT(300,LoadPerm.Max,5004);//197"

END_PROGRAM
```

### Package Logical/Automatic - Automatic sequencing

### Automatic.var - Package variables
```iecst
(********************************************************************
 * COPYRIGHT --
 ********************************************************************
 * Package: Automatic
 * File: Automatic.var
 * Author: nicke
 * Created: February, 2012
 ********************************************************************
 * Variables of package Automatic
 ********************************************************************)
VAR
	Belt1 : TrackProc; (*Belt timing control*)
	Belt2 : TrackProc; (*Belt timing control*)
	Belt3 : TrackProc; (*Belt timing control*)
	Belt4 : TrackProc; (*Belt timing control*)
	Belt5 : TrackProc; (*Belt timing control*)
	Belt6 : TrackProc; (*Belt timing control*)
	Belt7 : TrackProc; (*Belt timing control*)
	Belt8 : TrackProc; (*Belt timing control*)
END_VAR
```

### Program Logical/Automatic/ResetInv (IEC) - Reset Inverters Before scan

#### ResetInv.st - Implementation code
```iecst
(********************************************************************
 * COPYRIGHT --
 ********************************************************************
 * Program: ResetInv
 * File: ResetInv.st
 * Author: nicke
 ********************************************************************
 * Implementation of program ResetInv
 ********************************************************************)

PROGRAM _CYCLIC

    //INVERTER CL1 CONTROLS
    //SCALE DISPLAY VALUES OF M/MIN TO FREQUENCY FOR CONVEYOR SET SPEEDS
	CL1.Inv.Reference1[0].x := 00.0 ;
	CL1.Inv.Reference1[0].y := 00.0 ;
	CL1.Inv.Reference1[1].x := ScalePerm.CL1Scale ; //SPEED OF CONVEYOR AT 50HZ. ALTER AS REQUIRED
	CL1.Inv.Reference1[1].y    := 500.0 ;  //500 = 50HZ

	CASE InvPerms.CL1.Analog OF
		NO_ANALOG:
		VOLTAGE_TYPE_1:
			CL1.SpeedAnalog := ((INT_TO_REAL(CL1.Input.AI1R))/(AnalogPerm.CL1.V1.ActAnalog/AnalogPerm.CL1.V1.ActSpeed)) ;
		CURRENT_TYPE_1:
			CL1.SpeedAnalog := ((INT_TO_REAL(CL1.Input.AI3R))/(AnalogPerm.CL1.C1.ActAnalog/AnalogPerm.CL1.C1.ActSpeed)) ;
		CURRENT_TYPE_2:
			CL1.SpeedAnalog := ((INT_TO_REAL(CL1.Input.AI3R)-1638.4)/(AnalogPerm.CL1.C2.ActAnalog/AnalogPerm.CL1.C2.ActSpeed)) ; //1638.4 IS 4mA SHIFT FOR 4-20mA RANGE
		CL1.Inv.Reference1[1].y := 400.0 ; //REDUCE SCALE REFERENCE BY 20% TO ALLOW FOR 4mA SHIFT
	END_CASE
	CL1.SpeedAnalog := LIMIT(1, CL1.SpeedAnalog, 60) ;

	CL1.Inv.Scale1.NoOfPoints := 2 ;
	CL1.Inv.Scale1.ptr_table := ADR(CL1.Inv.Reference1)    ;

	//RESET INVERTER OUTPUTS BEFORE SCAN
	IF NOT(Control.Test) THEN
		memcpy(ADR(CL1.o),ADR(ClearInv),SIZEOF(ClearInv));
	END_IF

	//INVERTER ENABLE CONTROL
	IF(Control.Achieved1) OR(Control.Test) THEN
		IF(CL1.Input.ETAD_06) THEN
			CL1.Output.CMDD_01 := TRUE ;
			CL1.Output.CMDD_02 := TRUE ;
		END_IF
		IF(CL1.Input.ETAD_04) AND(CL1.Input.ETAD_05) THEN
			CL1.Output.CMDD_00 := TRUE ;
		END_IF
	END_IF

	//INVERTER RESET CONTROL
	IF NOT(Control.Achieved1) AND NOT(Control.Test) THEN
		CL1.Output.CMDD_00 := FALSE ;
		CL1.Output.CMDD_01 := FALSE ;
		CL1.Output.CMDD_02 := FALSE ;
		CL1.Output.CMDD_07 := FALSE ;
	END_IF

	//SET INVERTER FREQUENCY
	CL1.Inv.Scale1();
	CL1.o.SpeedRef := CL1.Inv.Scale1.y ;
	CL1.Output.LFR := REAL_TO_INT(CL1.o.SpeedRef) ;

	//INVERTER CS1 CONTROLS
	//SCALE DISPLAY VALUES OF M/MIN TO FREQUENCY FOR CONVEYOR SET SPEEDS
	CS1.Inv.Reference1[0].x := 00.0 ;
	CS1.Inv.Reference1[0].y := 00.0 ;
	CS1.Inv.Reference1[1].x := ScalePerm.CS1Scale ; //SPEED OF CONVEYOR AT 50HZ. ALTER AS REQUIRED
	CS1.Inv.Reference1[1].y    := 500.0 ;  //500 = 50HZ

	CASE InvPerms.CS1.Analog OF
		NO_ANALOG:
		VOLTAGE_TYPE_1:
			CS1.SpeedAnalog := ((INT_TO_REAL(CS1.Input.AI1R))/(AnalogPerm.CS1.V1.ActAnalog/AnalogPerm.CS1.V1.ActSpeed)) ;
		CURRENT_TYPE_1:
			CS1.SpeedAnalog := ((INT_TO_REAL(CS1.Input.AI3R))/(AnalogPerm.CS1.C1.ActAnalog/AnalogPerm.CS1.C1.ActSpeed)) ;
		CURRENT_TYPE_2:
			CS1.SpeedAnalog := ((INT_TO_REAL(CS1.Input.AI3R)-1638.4)/(AnalogPerm.CS1.C2.ActAnalog/AnalogPerm.CS1.C2.ActSpeed)) ; //1638.4 IS 4mA SHIFT FOR 4-20mA RANGE
		CS1.Inv.Reference1[1].y := 400.0 ; //REDUCE SCALE REFERENCE BY 20% TO ALLOW FOR 4mA SHIFT
	END_CASE
	CS1.SpeedAnalog := LIMIT(1, CS1.SpeedAnalog, 60) ;

	CS1.Inv.Scale1.NoOfPoints := 2 ;
	CS1.Inv.Scale1.ptr_table := ADR(CS1.Inv.Reference1)    ;

	//RESET INVERTER OUTPUTS BEFORE SCAN
	IF NOT(Control.Test) THEN
		memcpy(ADR(CS1.o),ADR(ClearInv),SIZEOF(ClearInv));
	END_IF

	//INVERTER ENABLE CONTROL
	IF(Control.Achieved1) OR(Control.Test) THEN
		IF(CS1.Input.ETAD_06) THEN
			CS1.Output.CMDD_01 := TRUE ;
			CS1.Output.CMDD_02 := TRUE ;
		END_IF
		IF(CS1.Input.ETAD_04) AND(CS1.Input.ETAD_05) THEN
			CS1.Output.CMDD_00 := TRUE ;
		END_IF
	END_IF

	//INVERTER RESET CONTROL
	IF NOT(Control.Achieved1) AND NOT(Control.Test) THEN
		CS1.Output.CMDD_00 := FALSE ;
		CS1.Output.CMDD_01 := FALSE ;
		CS1.Output.CMDD_02 := FALSE ;
		CS1.Output.CMDD_07 := FALSE ;
	END_IF

	//SET INVERTER FREQUENCY
	CS1.Inv.Scale1();
	CS1.o.SpeedRef := CS1.Inv.Scale1.y ;
	CS1.Output.LFR := REAL_TO_INT(CS1.o.SpeedRef) ;

	//INVERTER CV1 CONTROLS
	//SCALE DISPLAY VALUES OF M/MIN TO FREQUENCY FOR CONVEYOR SET SPEEDS
	CV1.Inv.Reference1[0].x := 00.0 ;
	CV1.Inv.Reference1[0].y := 00.0 ;
	CV1.Inv.Reference1[1].x := ScalePerm.CV1Scale ; //SPEED OF CONVEYOR AT 50HZ. ALTER AS REQUIRED
	CV1.Inv.Reference1[1].y    := 500.0 ;  //500 = 50HZ

	CASE InvPerms.CV1.Analog OF
		NO_ANALOG:
		VOLTAGE_TYPE_1:
			CV1.SpeedAnalog := ((INT_TO_REAL(CV1.Input.AI1R))/(AnalogPerm.CV1.V1.ActAnalog/AnalogPerm.CV1.V1.ActSpeed)) ;
		CURRENT_TYPE_1:
			CV1.SpeedAnalog := ((INT_TO_REAL(CV1.Input.AI3R))/(AnalogPerm.CV1.C1.ActAnalog/AnalogPerm.CV1.C1.ActSpeed)) ;
		CURRENT_TYPE_2:
			CV1.SpeedAnalog := ((INT_TO_REAL(CV1.Input.AI3R)-1638.4)/(AnalogPerm.CV1.C2.ActAnalog/AnalogPerm.CV1.C2.ActSpeed)) ; //1638.4 IS 4mA SHIFT FOR 4-20mA RANGE
		CV1.Inv.Reference1[1].y := 400.0 ; //REDUCE SCALE REFERENCE BY 20% TO ALLOW FOR 4mA SHIFT
	END_CASE
	CV1.SpeedAnalog := LIMIT(1, CV1.SpeedAnalog, 60) ;

	CV1.Inv.Scale1.NoOfPoints := 2 ;
	CV1.Inv.Scale1.ptr_table := ADR(CV1.Inv.Reference1)    ;

	//RESET INVERTER OUTPUTS BEFORE SCAN
	IF NOT(Control.Test) THEN
		memcpy(ADR(CV1.o),ADR(ClearInv),SIZEOF(ClearInv));
	END_IF

	//INVERTER ENABLE CONTROL
	IF(Control.Achieved1) OR(Control.Test) THEN
		IF(CV1.Input.ETAD_06) THEN
			CV1.Output.CMDD_01 := TRUE ;
			CV1.Output.CMDD_02 := TRUE ;
		END_IF
		IF(CV1.Input.ETAD_04) AND(CV1.Input.ETAD_05) THEN
			CV1.Output.CMDD_00 := TRUE ;
		END_IF
	END_IF

	//INVERTER RESET CONTROL
	IF NOT(Control.Achieved1) AND NOT(Control.Test) THEN
		CV1.Output.CMDD_00 := FALSE ;
		CV1.Output.CMDD_01 := FALSE ;
		CV1.Output.CMDD_02 := FALSE ;
		CV1.Output.CMDD_07 := FALSE ;
	END_IF

	//SET INVERTER FREQUENCY
	CV1.Inv.Scale1();
	CV1.o.SpeedRef := CV1.Inv.Scale1.y ;
	CV1.Output.LFR := REAL_TO_INT(CV1.o.SpeedRef) ;

	//INVERTER CC1 CONTROLS
	//SCALE DISPLAY VALUES OF M/MIN TO FREQUENCY FOR CONVEYOR SET SPEEDS
	CC1.Inv.Reference1[0].x := 00.0 ;
	CC1.Inv.Reference1[0].y := 00.0 ;
	CC1.Inv.Reference1[1].x := ScalePerm.CC1Scale ; //SPEED OF CONVEYOR AT 50HZ. ALTER AS REQUIRED
	CC1.Inv.Reference1[1].y    := 500.0 ;  //500 = 50HZ

	CASE InvPerms.CC1.Analog OF
		NO_ANALOG:
		VOLTAGE_TYPE_1:
			CC1.SpeedAnalog := ((INT_TO_REAL(CC1.Input.AI1R))/(AnalogPerm.CC1.V1.ActAnalog/AnalogPerm.CC1.V1.ActSpeed)) ;
		CURRENT_TYPE_1:
			CC1.SpeedAnalog := ((INT_TO_REAL(CC1.Input.AI3R))/(AnalogPerm.CC1.C1.ActAnalog/AnalogPerm.CC1.C1.ActSpeed)) ;
		CURRENT_TYPE_2:
			CC1.SpeedAnalog := ((INT_TO_REAL(CC1.Input.AI3R)-1638.4)/(AnalogPerm.CC1.C2.ActAnalog/AnalogPerm.CC1.C2.ActSpeed)) ; //1638.4 IS 4mA SHIFT FOR 4-20mA RANGE
		CC1.Inv.Reference1[1].y := 400.0 ; //REDUCE SCALE REFERENCE BY 20% TO ALLOW FOR 4mA SHIFT
	END_CASE
	CC1.SpeedAnalog := LIMIT(1, CC1.SpeedAnalog, 60) ;

	CC1.Inv.Scale1.NoOfPoints := 2 ;
	CC1.Inv.Scale1.ptr_table := ADR(CC1.Inv.Reference1)    ;

	//RESET INVERTER OUTPUTS BEFORE SCAN
	IF NOT(Control.Test) THEN
		memcpy(ADR(CC1.o),ADR(ClearInv),SIZEOF(ClearInv));
	END_IF

	//INVERTER ENABLE CONTROL
	IF(Control.Achieved1) OR(Control.Test) THEN
		IF(CC1.Input.ETAD_06) THEN
			CC1.Output.CMDD_01 := TRUE ;
			CC1.Output.CMDD_02 := TRUE ;
		END_IF
		IF(CC1.Input.ETAD_04) AND(CC1.Input.ETAD_05) THEN
			CC1.Output.CMDD_00 := TRUE ;
		END_IF
	END_IF

	//INVERTER RESET CONTROL
	IF NOT(Control.Achieved1) AND NOT(Control.Test) THEN
		CC1.Output.CMDD_00 := FALSE ;
		CC1.Output.CMDD_01 := FALSE ;
		CC1.Output.CMDD_02 := FALSE ;
		CC1.Output.CMDD_07 := FALSE ;
	END_IF

	//SET INVERTER FREQUENCY
	CC1.Inv.Scale1();
	CC1.o.SpeedRef := CC1.Inv.Scale1.y ;
	CC1.Output.LFR := REAL_TO_INT(CC1.o.SpeedRef) ;

	//INVERTER CC2 CONTROLS
	//SCALE DISPLAY VALUES OF M/MIN TO FREQUENCY FOR CONVEYOR SET SPEEDS
	CC2.Inv.Reference1[0].x := 00.0 ;
	CC2.Inv.Reference1[0].y := 00.0 ;
	CC2.Inv.Reference1[1].x := ScalePerm.CC2Scale ; //SPEED OF CONVEYOR AT 50HZ. ALTER AS REQUIRED
	CC2.Inv.Reference1[1].y    := 500.0 ;  //500 = 50HZ

	CASE InvPerms.CC2.Analog OF
		NO_ANALOG:
		VOLTAGE_TYPE_1:
			CC2.SpeedAnalog := ((INT_TO_REAL(CC2.Input.AI1R))/(AnalogPerm.CC2.V1.ActAnalog/AnalogPerm.CC2.V1.ActSpeed)) ;
		CURRENT_TYPE_1:
			CC2.SpeedAnalog := ((INT_TO_REAL(CC2.Input.AI3R))/(AnalogPerm.CC2.C1.ActAnalog/AnalogPerm.CC2.C1.ActSpeed)) ;
		CURRENT_TYPE_2:
			CC2.SpeedAnalog := ((INT_TO_REAL(CC2.Input.AI3R)-1638.4)/(AnalogPerm.CC2.C2.ActAnalog/AnalogPerm.CC2.C2.ActSpeed)) ; //1638.4 IS 4mA SHIFT FOR 4-20mA RANGE
		CC2.Inv.Reference1[1].y := 400.0 ; //REDUCE SCALE REFERENCE BY 20% TO ALLOW FOR 4mA SHIFT
	END_CASE
	CC2.SpeedAnalog := LIMIT(1, CC2.SpeedAnalog, 60) ;

	CC2.Inv.Scale1.NoOfPoints := 2 ;
	CC2.Inv.Scale1.ptr_table := ADR(CC2.Inv.Reference1)    ;

	//RESET INVERTER OUTPUTS BEFORE SCAN
	IF NOT(Control.Test) THEN
		memcpy(ADR(CC2.o),ADR(ClearInv),SIZEOF(ClearInv));
	END_IF

	//INVERTER ENABLE CONTROL
	IF(Control.Achieved1) OR(Control.Test) THEN
		IF(CC2.Input.ETAD_06) THEN
			CC2.Output.CMDD_01 := TRUE ;
			CC2.Output.CMDD_02 := TRUE ;
		END_IF
		IF(CC2.Input.ETAD_04) AND(CC2.Input.ETAD_05) THEN
			CC2.Output.CMDD_00 := TRUE ;
		END_IF
	END_IF

	//INVERTER RESET CONTROL
	IF NOT(Control.Achieved1) AND NOT(Control.Test) THEN
		CC2.Output.CMDD_00 := FALSE ;
		CC2.Output.CMDD_01 := FALSE ;
		CC2.Output.CMDD_02 := FALSE ;
		CC2.Output.CMDD_07 := FALSE ;
	END_IF

	//SET INVERTER FREQUENCY
	CC2.Inv.Scale1();
	CC2.o.SpeedRef := CC2.Inv.Scale1.y ;
	CC2.Output.LFR := REAL_TO_INT(CC2.o.SpeedRef) ;

	//INVERTER CS2 CONTROLS
	//SCALE DISPLAY VALUES OF M/MIN TO FREQUENCY FOR CONVEYOR SET SPEEDS
	CS2.Inv.Reference1[0].x := 00.0 ;
	CS2.Inv.Reference1[0].y := 00.0 ;
	CS2.Inv.Reference1[1].x := ScalePerm.CS2Scale ; //SPEED OF CONVEYOR AT 50HZ. ALTER AS REQUIRED
	CS2.Inv.Reference1[1].y    := 500.0 ;  //500 = 50HZ

	CASE InvPerms.CS2.Analog OF
		NO_ANALOG:
		VOLTAGE_TYPE_1:
			CS2.SpeedAnalog := ((INT_TO_REAL(CS2.Input.AI1R))/(AnalogPerm.CS2.V1.ActAnalog/AnalogPerm.CS2.V1.ActSpeed)) ;
		CURRENT_TYPE_1:
			CS2.SpeedAnalog := ((INT_TO_REAL(CS2.Input.AI3R))/(AnalogPerm.CS2.C1.ActAnalog/AnalogPerm.CS2.C1.ActSpeed)) ;
		CURRENT_TYPE_2:
			CS2.SpeedAnalog := ((INT_TO_REAL(CS2.Input.AI3R)-1638.4)/(AnalogPerm.CS2.C2.ActAnalog/AnalogPerm.CS2.C2.ActSpeed)) ; //1638.4 IS 4mA SHIFT FOR 4-20mA RANGE
		CS2.Inv.Reference1[1].y := 400.0 ; //REDUCE SCALE REFERENCE BY 20% TO ALLOW FOR 4mA SHIFT
	END_CASE
	CS2.SpeedAnalog := LIMIT(1, CS2.SpeedAnalog, 60) ;

	CS2.Inv.Scale1.NoOfPoints := 2 ;
	CS2.Inv.Scale1.ptr_table := ADR(CS2.Inv.Reference1)    ;

	//RESET INVERTER OUTPUTS BEFORE SCAN
	IF NOT(Control.Test) THEN
		memcpy(ADR(CS2.o),ADR(ClearInv),SIZEOF(ClearInv));
	END_IF

	//INVERTER ENABLE CONTROL
	IF(Control.Achieved1) OR(Control.Test) THEN
		IF(CS2.Input.ETAD_06) THEN
			CS2.Output.CMDD_01 := TRUE ;
			CS2.Output.CMDD_02 := TRUE ;
		END_IF
		IF(CS2.Input.ETAD_04) AND(CS2.Input.ETAD_05) THEN
			CS2.Output.CMDD_00 := TRUE ;
		END_IF
	END_IF

	//INVERTER RESET CONTROL
	IF NOT(Control.Achieved1) AND NOT(Control.Test) THEN
		CS2.Output.CMDD_00 := FALSE ;
		CS2.Output.CMDD_01 := FALSE ;
		CS2.Output.CMDD_02 := FALSE ;
		CS2.Output.CMDD_07 := FALSE ;
	END_IF

	//SET INVERTER FREQUENCY
	CS2.Inv.Scale1();
	CS2.o.SpeedRef := CS2.Inv.Scale1.y ;
	CS2.Output.LFR := REAL_TO_INT(CS2.o.SpeedRef) ;

	//INVERTER CV2 CONTROLS
	//SCALE DISPLAY VALUES OF M/MIN TO FREQUENCY FOR CONVEYOR SET SPEEDS
	CV2.Inv.Reference1[0].x := 00.0 ;
	CV2.Inv.Reference1[0].y := 00.0 ;
	CV2.Inv.Reference1[1].x := ScalePerm.CV2Scale ; //SPEED OF CONVEYOR AT 50HZ. ALTER AS REQUIRED
	CV2.Inv.Reference1[1].y    := 500.0 ;  //500 = 50HZ

	CASE InvPerms.CV2.Analog OF
		NO_ANALOG:
		VOLTAGE_TYPE_1:
			CV2.SpeedAnalog := ((INT_TO_REAL(CV2.Input.AI1R))/(AnalogPerm.CV2.V1.ActAnalog/AnalogPerm.CV2.V1.ActSpeed)) ;
		CURRENT_TYPE_1:
			CV2.SpeedAnalog := ((INT_TO_REAL(CV2.Input.AI3R))/(AnalogPerm.CV2.C1.ActAnalog/AnalogPerm.CV2.C1.ActSpeed)) ;
		CURRENT_TYPE_2:
			CV2.SpeedAnalog := ((INT_TO_REAL(CV2.Input.AI3R)-1638.4)/(AnalogPerm.CV2.C2.ActAnalog/AnalogPerm.CV2.C2.ActSpeed)) ; //1638.4 IS 4mA SHIFT FOR 4-20mA RANGE
		CV2.Inv.Reference1[1].y := 400.0 ; //REDUCE SCALE REFERENCE BY 20% TO ALLOW FOR 4mA SHIFT
	END_CASE
	CV2.SpeedAnalog := LIMIT(1, CV2.SpeedAnalog, 60) ;

	CV2.Inv.Scale1.NoOfPoints := 2 ;
	CV2.Inv.Scale1.ptr_table := ADR(CV2.Inv.Reference1)    ;

	//RESET INVERTER OUTPUTS BEFORE SCAN
	IF NOT(Control.Test) THEN
		memcpy(ADR(CV2.o),ADR(ClearInv),SIZEOF(ClearInv));
	END_IF

	//INVERTER ENABLE CONTROL
	IF(Control.Achieved1) OR(Control.Test) THEN
		IF(CV2.Input.ETAD_06) THEN
			CV2.Output.CMDD_01 := TRUE ;
			CV2.Output.CMDD_02 := TRUE ;
		END_IF
		IF(CV2.Input.ETAD_04) AND(CV2.Input.ETAD_05) THEN
			CV2.Output.CMDD_00 := TRUE ;
		END_IF
	END_IF

	//INVERTER RESET CONTROL
	IF NOT(Control.Achieved1) AND NOT(Control.Test) THEN
		CV2.Output.CMDD_00 := FALSE ;
		CV2.Output.CMDD_01 := FALSE ;
		CV2.Output.CMDD_02 := FALSE ;
		CV2.Output.CMDD_07 := FALSE ;
	END_IF

	//SET INVERTER FREQUENCY
	CV2.Inv.Scale1();
	CV2.o.SpeedRef := CV2.Inv.Scale1.y ;
	CV2.Output.LFR := REAL_TO_INT(CV2.o.SpeedRef) ;

	//INVERTER CC3 CONTROLS
	//SCALE DISPLAY VALUES OF M/MIN TO FREQUENCY FOR CONVEYOR SET SPEEDS
	CC3.Inv.Reference1[0].x := 00.0 ;
	CC3.Inv.Reference1[0].y := 00.0 ;
	CC3.Inv.Reference1[1].x := ScalePerm.CC3Scale ; //SPEED OF CONVEYOR AT 50HZ. ALTER AS REQUIRED
	CC3.Inv.Reference1[1].y    := 500.0 ;  //500 = 50HZ

	CASE InvPerms.CC3.Analog OF
		NO_ANALOG:
		VOLTAGE_TYPE_1:
			CC3.SpeedAnalog := ((INT_TO_REAL(CC3.Input.AI1R))/(AnalogPerm.CC3.V1.ActAnalog/AnalogPerm.CC3.V1.ActSpeed)) ;
		CURRENT_TYPE_1:
			CC3.SpeedAnalog := ((INT_TO_REAL(CC3.Input.AI3R))/(AnalogPerm.CC3.C1.ActAnalog/AnalogPerm.CC3.C1.ActSpeed)) ;
		CURRENT_TYPE_2:
			CC3.SpeedAnalog := ((INT_TO_REAL(CC3.Input.AI3R)-1638.4)/(AnalogPerm.CC3.C2.ActAnalog/AnalogPerm.CC3.C2.ActSpeed)) ; //1638.4 IS 4mA SHIFT FOR 4-20mA RANGE
		CC3.Inv.Reference1[1].y := 400.0 ; //REDUCE SCALE REFERENCE BY 20% TO ALLOW FOR 4mA SHIFT
	END_CASE
	CC3.SpeedAnalog := LIMIT(1, CC3.SpeedAnalog, 60) ;

	CC3.Inv.Scale1.NoOfPoints := 2 ;
	CC3.Inv.Scale1.ptr_table := ADR(CC3.Inv.Reference1)    ;

	//RESET INVERTER OUTPUTS BEFORE SCAN
	IF NOT(Control.Test) THEN
		memcpy(ADR(CC3.o),ADR(ClearInv),SIZEOF(ClearInv));
	END_IF

	//INVERTER ENABLE CONTROL
	IF(Control.Achieved1) OR(Control.Test) THEN
		IF(CC3.Input.ETAD_06) THEN
			CC3.Output.CMDD_01 := TRUE ;
			CC3.Output.CMDD_02 := TRUE ;
		END_IF
		IF(CC3.Input.ETAD_04) AND(CC3.Input.ETAD_05) THEN
			CC3.Output.CMDD_00 := TRUE ;
		END_IF
	END_IF

	//INVERTER RESET CONTROL
	IF NOT(Control.Achieved1) AND NOT(Control.Test) THEN
		CC3.Output.CMDD_00 := FALSE ;
		CC3.Output.CMDD_01 := FALSE ;
		CC3.Output.CMDD_02 := FALSE ;
		CC3.Output.CMDD_07 := FALSE ;
	END_IF

	//SET INVERTER FREQUENCY
	CC3.Inv.Scale1();
	CC3.o.SpeedRef := CC3.Inv.Scale1.y ;
	CC3.Output.LFR := REAL_TO_INT(CC3.o.SpeedRef) ;

	//INVERTER CC4 CONTROLS
	//SCALE DISPLAY VALUES OF M/MIN TO FREQUENCY FOR CONVEYOR SET SPEEDS
	CC4.Inv.Reference1[0].x := 00.0 ;
	CC4.Inv.Reference1[0].y := 00.0 ;
	CC4.Inv.Reference1[1].x := ScalePerm.CC4Scale ; //SPEED OF CONVEYOR AT 50HZ. ALTER AS REQUIRED
	CC4.Inv.Reference1[1].y    := 500.0 ;  //500 = 50HZ

	CASE InvPerms.CC4.Analog OF
		NO_ANALOG:
		VOLTAGE_TYPE_1:
			CC4.SpeedAnalog := ((INT_TO_REAL(CC4.Input.AI1R))/(AnalogPerm.CC4.V1.ActAnalog/AnalogPerm.CC4.V1.ActSpeed)) ;
		CURRENT_TYPE_1:
			CC4.SpeedAnalog := ((INT_TO_REAL(CC4.Input.AI3R))/(AnalogPerm.CC4.C1.ActAnalog/AnalogPerm.CC4.C1.ActSpeed)) ;
		CURRENT_TYPE_2:
			CC4.SpeedAnalog := ((INT_TO_REAL(CC4.Input.AI3R)-1638.4)/(AnalogPerm.CC4.C2.ActAnalog/AnalogPerm.CC4.C2.ActSpeed)) ; //1638.4 IS 4mA SHIFT FOR 4-20mA RANGE
		CC4.Inv.Reference1[1].y := 400.0 ; //REDUCE SCALE REFERENCE BY 20% TO ALLOW FOR 4mA SHIFT
	END_CASE
	CC4.SpeedAnalog := LIMIT(1, CC4.SpeedAnalog, 60) ;

	CC4.Inv.Scale1.NoOfPoints := 2 ;
	CC4.Inv.Scale1.ptr_table := ADR(CC4.Inv.Reference1)    ;

	//RESET INVERTER OUTPUTS BEFORE SCAN
	IF NOT(Control.Test) THEN
		memcpy(ADR(CC4.o),ADR(ClearInv),SIZEOF(ClearInv));
	END_IF

	//INVERTER ENABLE CONTROL
	IF(Control.Achieved1) OR(Control.Test) THEN
		IF(CC4.Input.ETAD_06) THEN
			CC4.Output.CMDD_01 := TRUE ;
			CC4.Output.CMDD_02 := TRUE ;
		END_IF
		IF(CC4.Input.ETAD_04) AND(CC4.Input.ETAD_05) THEN
			CC4.Output.CMDD_00 := TRUE ;
		END_IF
	END_IF

	//INVERTER RESET CONTROL
	IF NOT(Control.Achieved1) AND NOT(Control.Test) THEN
		CC4.Output.CMDD_00 := FALSE ;
		CC4.Output.CMDD_01 := FALSE ;
		CC4.Output.CMDD_02 := FALSE ;
		CC4.Output.CMDD_07 := FALSE ;
	END_IF

	//SET INVERTER FREQUENCY
	CC4.Inv.Scale1();
	CC4.o.SpeedRef := CC4.Inv.Scale1.y ;
	CC4.Output.LFR := REAL_TO_INT(CC4.o.SpeedRef) ;

	//INVERTER CB1 CONTROLS
	//SCALE DISPLAY VALUES OF M/MIN TO FREQUENCY FOR CONVEYOR SET SPEEDS
	CB1.Inv.Reference1[0].x := 00.0 ;
	CB1.Inv.Reference1[0].y := 00.0 ;
	CB1.Inv.Reference1[1].x := ScalePerm.CB1Scale ; //SPEED OF CONVEYOR AT 50HZ. ALTER AS REQUIRED
	CB1.Inv.Reference1[1].y    := 500.0 ;  //500 = 50HZ

	CASE InvPerms.CB1.Analog OF
		NO_ANALOG:
		VOLTAGE_TYPE_1:
			CB1.SpeedAnalog := ((INT_TO_REAL(CB1.Input.AI1R))/(AnalogPerm.CB1.V1.ActAnalog/AnalogPerm.CB1.V1.ActSpeed)) ;
		CURRENT_TYPE_1:
			CB1.SpeedAnalog := ((INT_TO_REAL(CB1.Input.AI3R))/(AnalogPerm.CB1.C1.ActAnalog/AnalogPerm.CB1.C1.ActSpeed)) ;
		CURRENT_TYPE_2:
			CB1.SpeedAnalog := ((INT_TO_REAL(CB1.Input.AI3R)-1638.4)/(AnalogPerm.CB1.C2.ActAnalog/AnalogPerm.CB1.C2.ActSpeed)) ; //1638.4 IS 4mA SHIFT FOR 4-20mA RANGE
		CB1.Inv.Reference1[1].y := 400.0 ; //REDUCE SCALE REFERENCE BY 20% TO ALLOW FOR 4mA SHIFT
	END_CASE
	CB1.SpeedAnalog := LIMIT(1, CB1.SpeedAnalog, 60) ;

	CB1.Inv.Scale1.NoOfPoints := 2 ;
	CB1.Inv.Scale1.ptr_table := ADR(CB1.Inv.Reference1)    ;

	//RESET INVERTER OUTPUTS BEFORE SCAN
	IF NOT(Control.Test) THEN
		memcpy(ADR(CB1.o),ADR(ClearInv),SIZEOF(ClearInv));
	END_IF

	//INVERTER ENABLE CONTROL
	IF(Control.Achieved1) OR(Control.Test) THEN
		IF(CB1.Input.ETAD_06) THEN
			CB1.Output.CMDD_01 := TRUE ;
			CB1.Output.CMDD_02 := TRUE ;
		END_IF
		IF(CB1.Input.ETAD_04) AND(CB1.Input.ETAD_05) THEN
			CB1.Output.CMDD_00 := TRUE ;
		END_IF
	END_IF

	//INVERTER RESET CONTROL
	IF NOT(Control.Achieved1) AND NOT(Control.Test) THEN
		CB1.Output.CMDD_00 := FALSE ;
		CB1.Output.CMDD_01 := FALSE ;
		CB1.Output.CMDD_02 := FALSE ;
		CB1.Output.CMDD_07 := FALSE ;
	END_IF

	//SET INVERTER FREQUENCY
	CB1.Inv.Scale1();
	CB1.o.SpeedRef := CB1.Inv.Scale1.y ;
	CB1.Output.LFR := REAL_TO_INT(CB1.o.SpeedRef) ;

	//INVERTER CB2 CONTROLS
	//SCALE DISPLAY VALUES OF M/MIN TO FREQUENCY FOR CONVEYOR SET SPEEDS
	CB2.Inv.Reference1[0].x := 00.0 ;
	CB2.Inv.Reference1[0].y := 00.0 ;
	CB2.Inv.Reference1[1].x := ScalePerm.CB2Scale ; //SPEED OF CONVEYOR AT 50HZ. ALTER AS REQUIRED
	CB2.Inv.Reference1[1].y    := 500.0 ;  //500 = 50HZ

	CASE InvPerms.CB2.Analog OF
		NO_ANALOG:
		VOLTAGE_TYPE_1:
			CB2.SpeedAnalog := ((INT_TO_REAL(CB2.Input.AI1R))/(AnalogPerm.CB2.V1.ActAnalog/AnalogPerm.CB2.V1.ActSpeed)) ;
		CURRENT_TYPE_1:
			CB2.SpeedAnalog := ((INT_TO_REAL(CB2.Input.AI3R))/(AnalogPerm.CB2.C1.ActAnalog/AnalogPerm.CB2.C1.ActSpeed)) ;
		CURRENT_TYPE_2:
			CB2.SpeedAnalog := ((INT_TO_REAL(CB2.Input.AI3R)-1638.4)/(AnalogPerm.CB2.C2.ActAnalog/AnalogPerm.CB2.C2.ActSpeed)) ; //1638.4 IS 4mA SHIFT FOR 4-20mA RANGE
		CB2.Inv.Reference1[1].y := 400.0 ; //REDUCE SCALE REFERENCE BY 20% TO ALLOW FOR 4mA SHIFT
	END_CASE
	CB2.SpeedAnalog := LIMIT(1, CB2.SpeedAnalog, 60) ;

	CB2.Inv.Scale1.NoOfPoints := 2 ;
	CB2.Inv.Scale1.ptr_table := ADR(CB2.Inv.Reference1)    ;

	//RESET INVERTER OUTPUTS BEFORE SCAN
	IF NOT(Control.Test) THEN
		memcpy(ADR(CB2.o),ADR(ClearInv),SIZEOF(ClearInv));
	END_IF

	//INVERTER ENABLE CONTROL
	IF(Control.Achieved1) OR(Control.Test) THEN
		IF(CB2.Input.ETAD_06) THEN
			CB2.Output.CMDD_01 := TRUE ;
			CB2.Output.CMDD_02 := TRUE ;
		END_IF
		IF(CB2.Input.ETAD_04) AND(CB2.Input.ETAD_05) THEN
			CB2.Output.CMDD_00 := TRUE ;
		END_IF
	END_IF

	//INVERTER RESET CONTROL
	IF NOT(Control.Achieved1) AND NOT(Control.Test) THEN
		CB2.Output.CMDD_00 := FALSE ;
		CB2.Output.CMDD_01 := FALSE ;
		CB2.Output.CMDD_02 := FALSE ;
		CB2.Output.CMDD_07 := FALSE ;
	END_IF

	//SET INVERTER FREQUENCY
	CB2.Inv.Scale1();
	CB2.o.SpeedRef := CB2.Inv.Scale1.y ;
	CB2.Output.LFR := REAL_TO_INT(CB2.o.SpeedRef) ;

	//INVERTER CRB CONTROLS
	//SCALE DISPLAY VALUES OF M/MIN TO FREQUENCY FOR CONVEYOR SET SPEEDS
	CRB.Inv.Reference1[0].x := 00.0 ;
	CRB.Inv.Reference1[0].y := 00.0 ;
	CRB.Inv.Reference1[1].x := ScalePerm.CRBScale ; //SPEED OF CONVEYOR AT 50HZ. ALTER AS REQUIRED
	CRB.Inv.Reference1[1].y    := 500.0 ;  //500 = 50HZ

	CASE InvPerms.CRB.Analog OF
		NO_ANALOG:
		VOLTAGE_TYPE_1:
			CRB.SpeedAnalog := ((INT_TO_REAL(CRB.Input.AI1R))/(AnalogPerm.CRB.V1.ActAnalog/AnalogPerm.CRB.V1.ActSpeed)) ;
		CURRENT_TYPE_1:
			CRB.SpeedAnalog := ((INT_TO_REAL(CRB.Input.AI3R))/(AnalogPerm.CRB.C1.ActAnalog/AnalogPerm.CRB.C1.ActSpeed)) ;
		CURRENT_TYPE_2:
			CRB.SpeedAnalog := ((INT_TO_REAL(CRB.Input.AI3R)-1638.4)/(AnalogPerm.CRB.C2.ActAnalog/AnalogPerm.CRB.C2.ActSpeed)) ; //1638.4 IS 4mA SHIFT FOR 4-20mA RANGE
		CRB.Inv.Reference1[1].y := 400.0 ; //REDUCE SCALE REFERENCE BY 20% TO ALLOW FOR 4mA SHIFT
	END_CASE
	CRB.SpeedAnalog := LIMIT(1, CRB.SpeedAnalog, 60) ;

	CRB.Inv.Scale1.NoOfPoints := 2 ;
	CRB.Inv.Scale1.ptr_table := ADR(CRB.Inv.Reference1)    ;

	//RESET INVERTER OUTPUTS BEFORE SCAN
	IF NOT(Control.Test) THEN
		memcpy(ADR(CRB.o),ADR(ClearInv),SIZEOF(ClearInv));
	END_IF

	//INVERTER ENABLE CONTROL
	IF(Control.Achieved1) OR(Control.Test) THEN
		IF(CRB.Input.ETAD_06) THEN
			CRB.Output.CMDD_01 := TRUE ;
			CRB.Output.CMDD_02 := TRUE ;
		END_IF
		IF(CRB.Input.ETAD_04) AND(CRB.Input.ETAD_05) THEN
			CRB.Output.CMDD_00 := TRUE ;
		END_IF
	END_IF

	//INVERTER RESET CONTROL
	IF NOT(Control.Achieved1) AND NOT(Control.Test) THEN
		CRB.Output.CMDD_00 := FALSE ;
		CRB.Output.CMDD_01 := FALSE ;
		CRB.Output.CMDD_02 := FALSE ;
		CRB.Output.CMDD_07 := FALSE ;
	END_IF

	//SET INVERTER FREQUENCY
	CRB.Inv.Scale1();
	CRB.o.SpeedRef := CRB.Inv.Scale1.y ;
	CRB.Output.LFR := REAL_TO_INT(CRB.o.SpeedRef) ;

	//INVERTER CRE CONTROLS
	//SCALE DISPLAY VALUES OF M/MIN TO FREQUENCY FOR CONVEYOR SET SPEEDS
	CRE.Inv.Reference1[0].x := 00.0 ;
	CRE.Inv.Reference1[0].y := 00.0 ;
	CRE.Inv.Reference1[1].x := ScalePerm.CREScale ; //SPEED OF CONVEYOR AT 50HZ. ALTER AS REQUIRED
	CRE.Inv.Reference1[1].y    := 500.0 ;  //500 = 50HZ

	CASE InvPerms.CRE.Analog OF
		NO_ANALOG:
		VOLTAGE_TYPE_1:
			CRE.SpeedAnalog := ((INT_TO_REAL(CRE.Input.AI1R))/(AnalogPerm.CRE.V1.ActAnalog/AnalogPerm.CRE.V1.ActSpeed)) ;
		CURRENT_TYPE_1:
			CRE.SpeedAnalog := ((INT_TO_REAL(CRE.Input.AI3R))/(AnalogPerm.CRE.C1.ActAnalog/AnalogPerm.CRE.C1.ActSpeed)) ;
		CURRENT_TYPE_2:
			CRE.SpeedAnalog := ((INT_TO_REAL(CRE.Input.AI3R)-1638.4)/(AnalogPerm.CRE.C2.ActAnalog/AnalogPerm.CRE.C2.ActSpeed)) ; //1638.4 IS 4mA SHIFT FOR 4-20mA RANGE
		CRE.Inv.Reference1[1].y := 400.0 ; //REDUCE SCALE REFERENCE BY 20% TO ALLOW FOR 4mA SHIFT
	END_CASE
	CRE.SpeedAnalog := LIMIT(1, CRE.SpeedAnalog, 60) ;

	CRE.Inv.Scale1.NoOfPoints := 2 ;
	CRE.Inv.Scale1.ptr_table := ADR(CRE.Inv.Reference1)    ;

	//RESET INVERTER OUTPUTS BEFORE SCAN
	IF NOT(Control.Test) THEN
		memcpy(ADR(CRE.o),ADR(ClearInv),SIZEOF(ClearInv));
	END_IF

	//INVERTER ENABLE CONTROL
	IF(Control.Achieved1) OR(Control.Test) THEN
		IF(CRE.Input.ETAD_06) THEN
			CRE.Output.CMDD_01 := TRUE ;
			CRE.Output.CMDD_02 := TRUE ;
		END_IF
		IF(CRE.Input.ETAD_04) AND(CRE.Input.ETAD_05) THEN
			CRE.Output.CMDD_00 := TRUE ;
		END_IF
	END_IF

	//INVERTER RESET CONTROL
	IF NOT(Control.Achieved1) AND NOT(Control.Test) THEN
		CRE.Output.CMDD_00 := FALSE ;
		CRE.Output.CMDD_01 := FALSE ;
		CRE.Output.CMDD_02 := FALSE ;
		CRE.Output.CMDD_07 := FALSE ;
	END_IF

	//SET INVERTER FREQUENCY
	CRE.Inv.Scale1();
	CRE.o.SpeedRef := CRE.Inv.Scale1.y ;
	CRE.Output.LFR := REAL_TO_INT(CRE.o.SpeedRef) ;

	//INVERTER CLB CONTROLS
	//SCALE DISPLAY VALUES OF M/MIN TO FREQUENCY FOR CONVEYOR SET SPEEDS
	CLB.Inv.Reference1[0].x := 00.0 ;
	CLB.Inv.Reference1[0].y := 00.0 ;
	CLB.Inv.Reference1[1].x := ScalePerm.CLBScale ; //SPEED OF CONVEYOR AT 50HZ. ALTER AS REQUIRED
	CLB.Inv.Reference1[1].y    := 500.0 ;  //500 = 50HZ

	CASE InvPerms.CLB.Analog OF
		NO_ANALOG:
		VOLTAGE_TYPE_1:
			CLB.SpeedAnalog := ((INT_TO_REAL(CLB.Input.AI1R))/(AnalogPerm.CLB.V1.ActAnalog/AnalogPerm.CLB.V1.ActSpeed)) ;
		CURRENT_TYPE_1:
			CLB.SpeedAnalog := ((INT_TO_REAL(CLB.Input.AI3R))/(AnalogPerm.CLB.C1.ActAnalog/AnalogPerm.CLB.C1.ActSpeed)) ;
		CURRENT_TYPE_2:
			CLB.SpeedAnalog := ((INT_TO_REAL(CLB.Input.AI3R)-1638.4)* 1.25) / ((((AnalogPerm.CLB.C2.ActAnalog)-1638.4)*1.25)/ AnalogPerm.CLB.C2.ActSpeed) ;
			//CLB.Inv.Reference1[1].y := 400.0 ; //REDUCE SCALE REFERENCE BY 20% TO ALLOW FOR 4mA SHIFT
	END_CASE
	CLB.SpeedAnalog := LIMIT(1, CLB.SpeedAnalog, 60) ;

	CLB.Inv.Scale1.NoOfPoints := 2 ;
	CLB.Inv.Scale1.ptr_table := ADR(CLB.Inv.Reference1)    ;

	//RESET INVERTER OUTPUTS BEFORE SCAN
	IF NOT(Control.Test) THEN
		memcpy(ADR(CLB.o),ADR(ClearInv),SIZEOF(ClearInv));
	END_IF

	//INVERTER ENABLE CONTROL
	IF(Control.Achieved1) OR(Control.Test) THEN
		IF(CLB.Input.ETAD_06) THEN
			CLB.Output.CMDD_01 := TRUE ;
			CLB.Output.CMDD_02 := TRUE ;
		END_IF
		IF(CLB.Input.ETAD_04) AND(CLB.Input.ETAD_05) THEN
			CLB.Output.CMDD_00 := TRUE ;
		END_IF
	END_IF

	//INVERTER RESET CONTROL
	IF NOT(Control.Achieved1) AND NOT(Control.Test) THEN
		CLB.Output.CMDD_00 := FALSE ;
		CLB.Output.CMDD_01 := FALSE ;
		CLB.Output.CMDD_02 := FALSE ;
		CLB.Output.CMDD_07 := FALSE ;
	END_IF

	//SET INVERTER FREQUENCY
	CLB.Inv.Scale1();
	CLB.o.SpeedRef := CLB.Inv.Scale1.y ;
	CLB.Output.LFR := REAL_TO_INT(CLB.o.SpeedRef) ;

	//RESET ALL .Inv.SCALE1.x FOR DISPLAY PURPOSES.
	CL1.Inv.Scale1.x   :=  0   ;
	CS1.Inv.Scale1.x   :=  0   ;
	CV1.Inv.Scale1.x   :=  0   ;
	CC1.Inv.Scale1.x   :=  0   ;
	CC2.Inv.Scale1.x   :=  0   ;
	CS2.Inv.Scale1.x   :=  0   ;
	CV2.Inv.Scale1.x   :=  0   ;
	CC3.Inv.Scale1.x   :=  0   ;
	CC4.Inv.Scale1.x   :=  0   ;
	CB1.Inv.Scale1.x   :=  0   ;
	CB2.Inv.Scale1.x   :=  0   ;
	CRB.Inv.Scale1.x   :=  0   ;
	CRE.Inv.Scale1.x   :=  0   ;
	CLB.Inv.Scale1.x   :=  0   ;

END_PROGRAM
```

### Program Logical/Automatic/AxBlocks (IEC)

#### Cyclic.st - Cyclic code
```iecst
PROGRAM _CYCLIC

	//BLOCK SEEK AND FIND OPERATION - AXIS 1
	Ax1.Blocks[0] := Track101.Active ;
	Ax1.Blocks[1] := Track102.Active ;
	Ax1.Blocks[2] := Track103.Active ;
	Ax1.Blocks[3] := Track104.Active ;
	Ax1.Blocks[8] := Control.ESClear ;
	Ax1.Blocks[9] := NOT(ArmsTemp1.DownDone) ;
	IF NOT(Control.Test) THEN
		Ax1.Blocks[10] := NOT(Ax1.OriginSet) ;
		Ax1.Blocks[11] := NOT(Control.Achieved1) ;
	ELSE
		Ax1.Blocks[10] := FALSE ;
		Ax1.Blocks[11] := FALSE ;
	END_IF

	//CHECK ARRAY FOR ON CONDITIONS
	FOR i:= 0 TO 12 DO
		IF Ax1.Blocks[i] = TRUE THEN
			Ax1.Block	:= 	TRUE	;
			EXIT							;
		ELSE
			Ax1.Block	:= 	FALSE	;
		END_IF
	END_FOR

	CASE Perms.HiVolume OF
		OFF:	// High Volume mode not selected
			Ax1.HiVol	:=	FALSE	;
		ON:		//High Volume mode selected
			IF EDGEPOS(Ax1.SeekFin) THEN
				Ax1.HiVol	:=	TRUE ;	//Latch On High Volume mode after first seek.
			END_IF
	END_CASE

	//BLOCK SEEK AND FIND OPERATION - AXIS 2
	Ax2.Blocks[0] := Track201.Active ;
	Ax2.Blocks[1] := Track202.Active ;
	Ax2.Blocks[2] := Track203.Active ;
	Ax2.Blocks[2] := Track204.Active ;
	Ax2.Blocks[8] := Control.ESClear ;
	Ax2.Blocks[9] := NOT(ArmsTemp2.DownDone) ;
	IF NOT(Control.Test) THEN
		Ax2.Blocks[10] := NOT(Ax2.OriginSet) ;
		Ax2.Blocks[11] := NOT(Control.Achieved1) ;
	ELSE
		Ax2.Blocks[10] := FALSE ;
		Ax2.Blocks[11] := FALSE ;
	END_IF
	Ax2.Blocks[12] := (S53Reed.In) OR NOT(S52Reed.In) ;

	//Check Array for conditions
	FOR i:= 0 TO 12 DO
		IF Ax2.Blocks[i] = TRUE THEN
			Ax2.Block	:= 	TRUE	;
			EXIT							;
		ELSE
			Ax2.Block	:= 	FALSE	;
		END_IF
	END_FOR

	CASE Perms.HiVolume OF
		OFF:	// High Volume mode not selected
			Ax2.HiVol	:=	FALSE	;
		ON:		//High Volume mode selected
			IF EDGEPOS(Ax2.SeekFin) THEN
				Ax2.HiVol	:=	TRUE ;	//Latch On High Volume mode after first seek.
			END_IF
	END_CASE

END_PROGRAM
```

### Program Logical/Automatic/ConLoad (IEC) - Loading Conveyor

#### ConLoadCyclic.st - Cyclic code
```iecst
(********************************************************************
 * COPYRIGHT --
 ********************************************************************
 * Program: ConLoad
 * File: ConLoadCyclic.st
 * Author: nicke
 ********************************************************************
 * Implementation of program ConLoad
 ********************************************************************)

PROGRAM _CYCLIC

   //TRACKINGSECTION END BLOCK CONDITIONS
	Tracking00.Blocks[0] := (Tracking10.Busy) ;
	Tracking00.Blocks[1] := ((Track011.Active) OR(Track012.Active)) AND(S56Lever.In) ;
	Tracking00.Blocks[2] := (CS1.Input.Fault) OR(CV1.Input.Fault) ;
	Tracking00.Blocks[3] := (CC1.Input.Fault) ;
	Tracking00.Blocks[4] := NOT(Sol31Pal2.Auto) ;
	Tracking00.Blocks[5] := NOT(Sol24DG1.Auto) ;
	Tracking00.Blocks[6] := NOT(SeamersII.DoneOUT[1]) ;
	Tracking00.Blocks[7] := NOT(ArmsTemp1.UpDone) ;
	Tracking00.Blocks[9] := (S3Photo.Int) ;
	Tracking00.Blocks[10] := (S4Photo.Int) ;
	Tracking00.Blocks[11] := NOT(S33Reed.In) ;
	Tracking00.Blocks[12] := (S50Reed.In) ;
	Tracking00.ControlIN := Control.Achieved1 ;
	Tracking00.EMOStart := EMO.StartLatch ;
	Tracking00.ESClear := Control.ESClear ;
	//Tracking00.BlockInhib := (Track912.Active) AND(S32Reed.In) AND NOT((Tracking00.Blocks[6]) OR(Tracking00.Blocks[7])) ;
	Tracking00 ();
	Tracking00.ResMan := FALSE ;
	//RESET OF OUTPUTS
	Sol30Pal1.Auto := FALSE ;
	Sol40Datum.Auto := FALSE ;
	Ax1.RaiseArms := FALSE ;
	CASE Tracking00.Index OF
		0: //RESET ALL TRACKBIT FOR SELECTED TRACKINGSECTION
			Track001 := TrackClear ;
			Track002 := TrackClear ;
			Track003 := TrackClear ;
			Track004 := TrackClear ;
			Track005 := TrackClear ;
			//START CONDITION FOR LOADING
			IF((S45Foot.In) AND(S30Reed.In) AND NOT(Tracking90.Busy) AND(Control.Achieved1)) THEN
				Tracking00.IndexIN := 1 ;
			END_IF
		1: //TRACK FROM S45Foot.In (P) TO S31Reed.In (P)
			Track002 := TrackClear ;
			Track003 := TrackClear ;
			Track004 := TrackClear ;
			Track005 := TrackClear ;
			//FB INPUTS
			Track001.FixedIN := Tracking00.FixedOUT ;
			Track001.TimeoutEN := TRUE ;
			Track001.TimeoutACK := Warn.Ack ;
			Track001.TimeoutBlock := (Warn.Block) ;
			Track001.DelayPT := TrackDelayPT.PTTrack001 ;
			//FB CALL
			Track001 ();
			//FB OUTPUTS
			Sol30Pal1.Auto := (Track001.SolOUT) ;
			IF(Track001.Done) THEN
				Tracking00.IndexIN := 2 ;
			END_IF
		2: //TRACK FROM S31Reed.In (P) TO S1Photo.Int (P)
			Track001 := TrackClear ;
			Track003 := TrackClear ;
			Track004 := TrackClear ;
			Track005 := TrackClear ;
			//FB INPUTS
			Track002.FixedIN := Tracking00.FixedOUT ;
			Track002.Speed := Speeds.SpeedTrans ;
			Track002.TimeoutEN := TRUE ;
			Track002.DelayPT := TrackDelayPT.PTTrack002 ;
			//FB CALL
			Track002 ();
			//FB OUTPUTS
			CL1.o.Run[0] := Track002.RunOUT ;
			CL1.Inv.Scale1.x := Track002.SpeedOUT ;
			Sol30Pal1.Auto := (Track002.SolOUT) ;
			IF(Track002.TimeoutOUT) THEN
				Tracking00.IndexIN := 0 ;
			END_IF
			IF(Track002.Done) THEN
				Tracking00.IndexIN := 3 ;
				Tracking00.RowBlockIN := FurnaceSelect.Selected; //Input for Furnace 2 selection
			END_IF
		3: //TRACK FROM S1Photo.Int (P) TO S2Photo.Int (P)
			Track001 := TrackClear ;
			Track002 := TrackClear ;
			Track004 := TrackClear ;
			Track005 := TrackClear ;
			//FB INPUTS
			Track003.FixedIN := Tracking00.FixedOUT ;
			IF(S56Lever.In) THEN
				Track003.Speed := Speeds.SpeedLaser ;
			ELSE
				Track003.Speed := Speeds.SpeedSlow ;
			END_IF
			Track003.TimeoutEN := TRUE ;
			Track003.TimeoutACK := Warn.Ack ;
			Track003.TimeoutBlock := (Warn.Block) ;
			Track003.DelayPT := TrackDelayPT.PTTrack003 ;
			//FB CALL
			Track003 ();
			//FB OUTPUTS
			CL1.o.Run[0] := Track003.RunOUT ;
			CL1.Inv.Scale1.x := Track003.SpeedOUT ;
			Sol30Pal1.Auto := (Track003.SolOUT) ;
			IF(Track003.Done) THEN
				Tracking00.IndexIN := 4 ;
				IF(S56Lever.In) THEN
					Tracking01.IndexIN := 1 ;
				END_IF
			END_IF
		4: //TRACK FROM S2Photo.Int (P) TO Ax1.SeekFin (P)
			Track001 := TrackClear ;
			Track002 := TrackClear ;
			Track003 := TrackClear ;
			Track005 := TrackClear ;
			//FB INPUTS
			Track004.FixedIN := Tracking00.FixedOUT ;
			//FB CALL
			Track004 ();
			//FB OUTPUTS
			Sol30Pal1.Auto := (Track004.SolOUT) ;
			IF NOT(Ax1.HiVol) THEN
				Ax1.Seek1 := (Track004.SolOUT) AND NOT(Ax1.Block) ;
			ELSE
				Tracking00.IndexIN := 5 ;
			END_IF
			IF(Track004.Done) THEN
				Tracking00.IndexIN := 5 ;
			END_IF
		5: //TRACK FROM Ax1.SeekFin (P) TO NOT Tracking00.Blocked (-)
			Track001 := TrackClear ;
			Track002 := TrackClear ;
			Track003 := TrackClear ;
			Track004 := TrackClear ;
			//FB INPUTS
			Track005.FixedIN := Tracking00.FixedOUT ;
			//FB CALL
			Track005 ();
			//FB OUTPUTS
			Sol30Pal1.Auto := (Track005.SolOUT) ;
			Ax1.RaiseArms := (Track005.SolOUT) ;
			IF(Track005.Done) THEN
				Tracking00.IndexIN := 0 ;
				Tracking10.IndexIN := 1 ;
				Tracking10.RowBlockIN := Tracking00.RowBlock ;
				Tracking90.IndexIN := 1 ;
			END_IF
	END_CASE

	//TRACKBIT DONE CONDITIONS
	Track001.DoneIN := EDGEPOS(S31Reed.In) ;
	Track002.DoneIN := EDGEPOS(S1Photo.Int) ;
	Track003.DoneIN := EDGEPOS(S2Photo.Int) ;
	Track004.DoneIN := EDGEPOS(Ax1.SeekFin) ;
	Track005.DoneIN := NOT(Tracking00.Blocked) ;

	Ax1.Active := Track004.Active ;

	//TRACKINGSECTION END BLOCK CONDITIONS
	Tracking90.ControlIN := Control.Achieved1 ;
	Tracking90.EMOStart := EMO.StartLatch ;
	Tracking90.ESClear := Control.ESClear ;
	Tracking90 ();
	Tracking90.ResMan := FALSE ;
	CASE Tracking90.Index OF
		0: //RESET ALL TRACKBIT FOR SELECTED TRACKINGSECTION
			Track901 := TrackClear ;
		1: //TRACK FROM NOT Tracking00.Blocked (-) TO S2Photo.Int (N)
			//FB INPUTS
			Track901.FixedIN := Tracking90.FixedOUT ;
			Track901.RunBlock := (Track101.TimeoutOUT) OR(Track104.TimeoutOUT) OR NOT((Track101.RunOUT) OR(Track104.RunOUT)) ;
			IF (ProcessMode.In) THEN
				Track901.Speed := Speeds.SpeedSeamSlow;
			ELSE
				Track901.Speed := Speeds.SpeedSeam ;
			END_IF
			//FB CALL
			Track901 ();
			//FB OUTPUTS
			CL1.o.Run[0] := Track901.RunOUT ;
			CL1.Inv.Scale1.x := Track901.SpeedOUT ;
			Sol30Pal1.Auto := (Track901.SolOUT) ;
			IF(Track901.Done) THEN
				Tracking90.IndexIN := 0 ;
			END_IF
	END_CASE

	//TRACKBIT DONE CONDITIONS
	Track901.DoneIN := EDGENEG(S2Photo.Int) ;

	//MANUAL RESET CONDITIONS FOR CONCURRENT TRACKBIT
	Tracking90.ResMan := Tracking10.ResMan ;
	IF(Tracking10.IndexIN = 0) THEN
		Tracking90.IndexIN := 0 ;
	END_IF

	//TRACKINGSECTION END BLOCK CONDITIONS
	Tracking01.Blocks[1] := Track005.Active ;
	Tracking01.ControlIN := Control.Achieved1 ;
	Tracking01.EMOStart := EMO.StartLatch ;
	Tracking01.ESClear := Control.ESClear ;
	Tracking01 ();
	Tracking01.ResMan := FALSE ;
	//RESET OF OUTPUTS
	LaserFire.Auto := FALSE ;
	Sol35Laser.Auto := Control.Achieved1 ;
	CASE Tracking01.Index OF
		0: //RESET ALL TRACKBIT FOR SELECTED TRACKINGSECTION
			Track011 := TrackClear ;
			Track012 := TrackClear ;
			Track013 := TrackClear ;
		1: //TRACK FROM S2Photo.Int (P) TO Track011.DelayTON.Q (-)
			Track012 := TrackClear ;
			Track013 := TrackClear ;
			//FB INPUTS
			Track011.FixedIN := Tracking01.FixedOUT ;
			Track011.TrackDelayEN := TRUE ;
			Track011.DelayPT := TrackDelayPT.PTTrack011 ;
			//FB CALL
			Track011 ();
			//FB OUTPUTS
			IF(Track011.Done) THEN
				Tracking01.IndexIN := 2 ;
			END_IF
		2: //TRACK FROM Track011.DelayTON.Q (-) TO LaserBusy.In (N)
			Track011 := TrackClear ;
			Track013 := TrackClear ;
			//FB INPUTS
			Track012.FixedIN := Tracking01.FixedOUT ;
			Track012.DelayPT := 1200 ;
			//FB CALL
			Track012 ();
			//FB OUTPUTS
			LaserFire.Auto := (Track012.SolOUT) ;
			IF(Track012.Done) THEN
				Tracking01.IndexIN := 3 ;
			END_IF
			IF(Track012.TimeoutOUT) THEN
				Tracking01.IndexIN := 3 ;
			END_IF
		3: //TRACK FROM LaserBusy.In (N) TO NOT Tracking01.Blocked (-)
			Track011 := TrackClear ;
			Track012 := TrackClear ;
			//FB INPUTS
			Track013.FixedIN := Tracking01.FixedOUT ;
			//FB CALL
			Track013 ();
			//FB OUTPUTS
			IF(Track013.Done) THEN
				Tracking01.IndexIN := 0 ;
			END_IF
	END_CASE

	//TRACKBIT DONE CONDITIONS
	//Track012.DoneIN := EDGENEG(LaserBusy.In) ;
	IF EDGENEG(LaserBusy.In) AND(Track012.Active) THEN
		Track012.TimeoutEN := TRUE ;
	END_IF
	Track013.DoneIN := NOT(Tracking01.Blocked) ;

	//MANUAL RESET CONDITIONS FOR CONCURRENT TRACKBIT
	Tracking01.ResMan := FALSE ;
	IF(Tracking00.IndexIN = 0) THEN
		IF(Tracking10.ResMan) THEN
			Tracking01.ResMan := TRUE ;
		END_IF
	END_IF
	IF EDGENEG(S56Lever.In) THEN
		Tracking01.ResMan := TRUE ;
	END_IF

END_PROGRAM
```

### Program Logical/Automatic/ConSeam1 (IEC) - Seaming 1 Conveyor

#### ConSeam1Cyclic.st - Cyclic code
```iecst
(********************************************************************
 * COPYRIGHT --
 ********************************************************************
 * PROGRAM: ConSeam1
 * File: ConSeam1Cyclic.st
 * Author: nicke
 ********************************************************************
 * Implementation OF PROGRAM ConSeam1
 ********************************************************************)

PROGRAM _CYCLIC

   //TRACKINGSECTION END BLOCK CONDITIONS
	Tracking10.Blocks[0] := (Tracking11.Busy) ;
	Tracking10.Blocks[1] := (Tracking91.Busy) ;
	Tracking10.Blocks[2] := (CC2.Input.Fault) ;
	Tracking10.Blocks[3] := (CS2.Input.Fault) OR(CV2.Input.Fault) ;
	Tracking10.Blocks[9] := (S5Photo.Int) ;
	Tracking10.Blocks[10] := (S6Photo.Int) ;
	Tracking10.Blocks[11] := (S7Photo.Int) ;
	Tracking10.ControlIN := Control.Achieved1 ;
	Tracking10.EMOStart := EMO.StartLatch ;
	Tracking10.ESClear := Control.ESClear ;
	Tracking10 ();
	Tracking10.ResMan := FALSE ;
	//RESET OF OUTPUTS
	Seaming.Start1 := FALSE ;
	Seaming.Stop1 := FALSE ;
	Sol24DG1.Auto := TRUE ;
	Sol24DG1B.Auto := FALSE ;
	Sol31Pal2.Auto := TRUE ;
	CASE Tracking10.Index OF
		0: //RESET ALL TRACKBIT FOR SELECTED TRACKINGSECTION
			Track101 := TrackClear ;
			Track102 := TrackClear ;
			Track103 := TrackClear ;
			Track104 := TrackClear ;
			Track105 := TrackClear ;
			Track106 := TrackClear ;
			Track107 := TrackClear ;
			Track108 := TrackClear ;
		1: //TRACK FROM NOT Tracking00.Blocked (-) TO S4Photo.Int (P)
			Track102 := TrackClear ;
			Track103 := TrackClear ;
			Track104 := TrackClear ;
			Track105 := TrackClear ;
			Track106 := TrackClear ;
			Track107 := TrackClear ;
			Track108 := TrackClear ;
			//FB INPUTS
			Track101.FixedIN := Tracking10.FixedOUT ;
			IF (ProcessMode.In) THEN
				Track101.Speed := Speeds.SpeedSeamSlow;
			ELSE
				Track101.Speed := Speeds.SpeedSeam ;
			END_IF
			Track101.RunBlock := NOT(SeamersII.DoneOUT[1]) ;
			Track101.TimeoutEN := TRUE ;
			Track101.TimeoutACK := Warn.Ack ;
			Track101.TimeoutBlock := (Warn.Block) ;
			Track101.DelayPT := TrackDelayPT.PTTrack101 ;
			//FB CALL
			Track101 ();
			//FB OUTPUTS
			CS1.o.Run[0] := Track101.RunOUT ;
			CV1.o.Run[0] := Track101.RunOUT ;
			CC1.o.Run[0] := Track101.RunOUT ;
			CS1.Inv.Scale1.x := Track101.SpeedOUT ;
			CV1.Inv.Scale1.x := Track101.SpeedOUT ;
			CC1.Inv.Scale1.x := Track101.SpeedOUT ;
			Ax1.RaiseArms := (Track101.SolOUT) ;
			IF(Track101.Done) THEN
				Tracking10.IndexIN := 4 ;
				Tracking10.LengthIN := Ax1.Measure/10.0 ;
			END_IF
		2: //TRACK FROM S3Photo.Int (P) TO S3Photo.Int (N)
			Track101 := TrackClear ;
			Track103 := TrackClear ;
			Track104 := TrackClear ;
			Track105 := TrackClear ;
			Track106 := TrackClear ;
			Track107 := TrackClear ;
			Track108 := TrackClear ;
			//FB INPUTS
//			Track102.FixedIN := Tracking10.FixedOUT ;
//			IF (ProcessMode.In) THEN
//				Track102.Speed := Speeds.SpeedSeamSlow;
//			ELSE
//				Track102.Speed := Speeds.SpeedSeam ;
//			END_IF
//			Track102.RunBlock := NOT(SeamersII.DoneOUT[1]) ;
//			Track102.TimeoutEN := TRUE ;
//			Track102.TimeoutACK := Warn.Ack ;
//			Track102.TimeoutBlock := (Warn.Block) ;
//			Track102.DelayPT := TrackDelayPT.PTTrack102 ;
//			//FB CALL
//			Track102 ();
//			//FB OUTPUTS
//			CS1.o.Run[0] := Track102.RunOUT ;
//			CV1.o.Run[0] := Track102.RunOUT ;
//			CC1.o.Run[0] := Track102.RunOUT ;
//			CS1.Inv.Scale1.x := Track102.SpeedOUT ;
//			CV1.Inv.Scale1.x := Track102.SpeedOUT ;
//			CC1.Inv.Scale1.x := Track102.SpeedOUT ;
//			Seaming.Start1 := (Track102.SolOUT) ;
//			Ax1.RaiseArms := (Track102.SolOUT) ;
//			IF(Track102.Done) THEN
//				Tracking10.IndexIN := 3 ;
//			END_IF
		3: //TRACK FROM S3Photo.Int (N) TO Belts1.Done (P)
			Track101 := TrackClear ;
			Track102 := TrackClear ;
			Track104 := TrackClear ;
			Track105 := TrackClear ;
			Track106 := TrackClear ;
			Track107 := TrackClear ;
			Track108 := TrackClear ;
			//FB INPUTS
//			Track103.FixedIN := Tracking10.FixedOUT ;
//			IF (ProcessMode.In) THEN
//				Track103.Speed := Speeds.SpeedSeamSlow;
//			ELSE
//				Track103.Speed := Speeds.SpeedSeam ;
//			END_IF
//			Track103.RunBlock := NOT(SeamersII.DoneOUT[1]) ;
//			//FB CALL
//			Track103 ();
//			//FB OUTPUTS
//			CS1.o.Run[0] := Track103.RunOUT ;
//			CV1.o.Run[0] := Track103.RunOUT ;
//			CC1.o.Run[0] := Track103.RunOUT ;
//			CS1.Inv.Scale1.x := Track103.SpeedOUT ;
//			CV1.Inv.Scale1.x := Track103.SpeedOUT ;
//			CC1.Inv.Scale1.x := Track103.SpeedOUT ;
//			Seaming.Stop1 := (Track103.SolOUT) ;
//			Ax1.RaiseArms := (Track103.SolOUT) ;
//			IF(Track103.Done) THEN
//				Tracking10.IndexIN := 4 ;
//				Tracking10.LengthIN := Ax1.Measure/10.0 ;
//			END_IF
		4: //TRACK FROM S4Photo.int (P) TO S4Photo.Int (N)
			Track101 := TrackClear ;
			Track102 := TrackClear ;
			Track103 := TrackClear ;
			Track105 := TrackClear ;
			Track106 := TrackClear ;
			Track107 := TrackClear ;
			Track108 := TrackClear ;
			//FB INPUTS
			Track104.FixedIN := Tracking10.FixedOUT ;
			IF (ProcessMode.In) THEN
				Track104.Speed := Speeds.SpeedSeamSlow;
			ELSE
				Track104.Speed := Speeds.SpeedSeam ;
			END_IF
			Track104.TimeoutEN := TRUE ;
			Track104.TimeoutACK := Warn.Ack ;
			Track104.TimeoutBlock := (Warn.Block) ;
			Track104.DelayPT := TrackDelayPT.PTTrack104 ;
			//FB CALL
			Track104 ();
			//FB OUTPUTS
			CS1.o.Run[0] := Track104.RunOUT ;
			CV1.o.Run[0] := Track104.RunOUT ;
			CC1.o.Run[0] := Track104.RunOUT ;
			CS1.Inv.Scale1.x := Track104.SpeedOUT ;
			CV1.Inv.Scale1.x := Track104.SpeedOUT ;
			CC1.Inv.Scale1.x := Track104.SpeedOUT ;
			Ax1.RaiseArms := (Track104.SolOUT) ;
			IF(Track104.Done) THEN
				Tracking10.IndexIN := 5 ;
			END_IF
		5: //TRACK FROM S4Photo.Int (N) TO Track105.DelayTON.Q (P)
			Track101 := TrackClear ;
			Track102 := TrackClear ;
			Track103 := TrackClear ;
			Track104 := TrackClear ;
			Track106 := TrackClear ;
			Track107 := TrackClear ;
			Track108 := TrackClear ;
			//FB INPUTS
			Track105.FixedIN := Tracking10.FixedOUT ;
			Track105.Speed := Speeds.SpeedSlow ;
			Track105.TrackDelayEN := TRUE ;
			Track105.DelayPT := TrackDelayPT.PTTrack105 ;
			//FB CALL
			Track105 ();
			//FB OUTPUTS
			CC1.o.Run[0] := Track105.RunOUT ;
			CC1.Inv.Scale1.x := Track105.SpeedOUT ;
			IF(Track105.Done) THEN
				Tracking10.IndexIN := 6 ;
			END_IF
		6: //TRACK FROM Track105.DelayTON.Q (P) TO S50Reed.In (P)
			Track101 := TrackClear ;
			Track102 := TrackClear ;
			Track103 := TrackClear ;
			Track104 := TrackClear ;
			Track105 := TrackClear ;
			Track107 := TrackClear ;
			Track108 := TrackClear ;
			//FB INPUTS
			Track106.FixedIN := Tracking10.FixedOUT ;
			Track106.TimeoutEN := TRUE ;
			Track106.TimeoutACK := Warn.Ack ;
			Track106.TimeoutBlock := (Warn.Block) ;
			Track106.DelayPT := TrackDelayPT.PTTrack106 ;
			//FB CALL
			Track106 ();
			//FB OUTPUTS
			Sol24DG1B.Auto := (Track106.SolOUT) ;
			IF(Track106.Done) THEN
				Tracking10.IndexIN := 7 ;
			END_IF
		7: //TRACK FROM S50Reed.In (P) TO Track107.DelayTON.Q (P)
			Track101 := TrackClear ;
			Track102 := TrackClear ;
			Track103 := TrackClear ;
			Track104 := TrackClear ;
			Track105 := TrackClear ;
			Track106 := TrackClear ;
			Track108 := TrackClear ;
			//FB INPUTS
			Track107.FixedIN := Tracking10.FixedOUT ;
			Track107.Speed := Speeds.SpeedSlow ;
			Track107.TrackDelayEN := TRUE ;
			Track107.DelayPT := TrackDelayPT.PTTrack107 ;
			//FB CALL
			Track107 ();
			//FB OUTPUTS
			CC1.o.Rev[0] := Track107.RunOUT ;
			CC1.Inv.Scale1.x := Track107.SpeedOUT ;
			Sol24DG1B.Auto := (Track107.SolOUT) ;
			IF(Track107.Done) THEN
				Tracking10.IndexIN := 8 ;
			END_IF
		8: //TRACK FROM Track107.DelayTON.Q (P) TO NOT Tracking10.Blocked (-)
			Track101 := TrackClear ;
			Track102 := TrackClear ;
			Track103 := TrackClear ;
			Track104 := TrackClear ;
			Track105 := TrackClear ;
			Track106 := TrackClear ;
			Track107 := TrackClear ;
			//FB INPUTS
			Track108.FixedIN := Tracking10.FixedOUT ;
			//FB CALL
			Track108 ();
			//FB OUTPUTS
			Sol24DG1B.Auto := (Track108.SolOUT) ;
			IF(Track108.Done) THEN
				Tracking10.IndexIN := 0 ;
				Tracking11.IndexIN := 1 ;
				Tracking91.IndexIN := 1 ;
				Tracking11.LengthIN := Tracking10.Length ;
				Tracking11.RowBlockIN := Tracking10.RowBlock ;
			END_IF
	END_CASE

	//TRACKBIT DONE CONDITIONS
	Track101.DoneIN := EDGEPOS(S4Photo.Int) ;
//	Track102.DoneIN := EDGENEG(S3Photo.Int) ;
//	Track103.DoneIN := EDGEPOS(Belts1.Done) ;
	Track104.DoneIN := EDGENEG(S4Photo.Int) ;
	Track106.DoneIN := EDGEPOS(S50Reed.In) ;
	Track108.DoneIN := NOT(Tracking10.Blocked) ;

	//TRACKINGSECTION END BLOCK CONDITIONS
	Tracking91.ControlIN := Control.Achieved1 ;
	Tracking91.EMOStart := EMO.StartLatch ;
	Tracking91.ESClear := Control.ESClear ;
	Tracking91 ();
	Tracking91.ResMan := FALSE ;
	CASE Tracking91.Index OF
		0: //RESET ALL TRACKBIT FOR SELECTED TRACKINGSECTION
			Track911 := TrackClear ;
			Track912 := TrackClear ;
		1: //TRACK FROM NOT Tracking11.Blocked (-) TO NOT S9Photo.Int (-)
			Track912 := TrackClear ;
			//FB INPUTS
			Track911.FixedIN := Tracking91.FixedOUT ;
			//FB CALL
			Track911 ();
			//FB OUTPUTS
			Sol24DG1.Auto := NOT(Track911.SolOUT) ;
			Sol24DG1B.Auto := (Track911.SolOUT) ;
			Sol31Pal2.Auto := NOT(Track911.SolOUT) ;
			IF(Track911.Done) THEN
				Tracking91.IndexIN := 2 ;
			END_IF
		2: //TRACK FROM NOT S9Photo.Int (-) TO S5Photo.Int (N)
			Track911 := TrackClear ;
			//FB INPUTS
			Track912.FixedIN := Tracking91.FixedOUT ;
			//FB CALL
			Track912 ();
			//FB OUTPUTS
			Sol24DG1.Auto := NOT(Track912.SolOUT) ;
			Sol24DG1B.Auto := (Track912.SolOUT) ;
			Sol31Pal2.Auto := NOT(Track912.SolOUT) ;
			IF(Track912.Done) THEN
				Tracking91.IndexIN := 0 ;
			END_IF
	END_CASE

	//TRACKBIT DONE CONDITIONS
	Track911.DoneIN := NOT(S9Photo.Int) ;
	Track912.DoneIN := EDGENEG(S5Photo.Int) ;

	//MANUAL RESET CONDITIONS FOR CONCURRENT TRACKBIT
	Tracking91.ResMan := (Tracking11.ResMan) OR((Tracking20.ResMan) AND((Track201.Active) OR(Track202.Active))) ;
	IF(Tracking11.IndexIN = 0) AND NOT((Track201.Active) OR(Track202.Active)) THEN
		Tracking91.IndexIN := 0 ;
	END_IF

END_PROGRAM
```

### Program Logical/Automatic/ConCorner (IEC) - Corner Conveyor Control

#### ConCornerCyclic.st - Cyclic code
```iecst
(********************************************************************
 * COPYRIGHT --
 ********************************************************************
 * PROGRAM: ConCorner
 * File: ConCornerCyclic.st
 * Author: NickE
 ********************************************************************
 * Implementation OF PROGRAM ConCorner
 ********************************************************************)

PROGRAM _CYCLIC

   //TRACKINGSECTION END BLOCK CONDITIONS
	Tracking11.Blocks[0] := (Tracking20.Busy) ;
	Tracking11.Blocks[1] := (Track301.Active) ;
	Tracking11.Blocks[2] := (CS2.Input.Fault) OR(CV2.Input.Fault) ;
	Tracking11.Blocks[3] := (CC3.Input.Fault) ;
	Tracking11.Blocks[4] := (Sol32Pal3.Auto) ;
	Tracking11.Blocks[6] := NOT(SeamersII.DoneOUT[2]) ;
	Tracking11.Blocks[7] := NOT(ArmsTemp2.UpDone) ;
	Tracking11.Blocks[9] := (S8Photo.Int) ;
	Tracking11.Blocks[10] := (S12Photo.Int) ;
	Tracking11.Blocks[11] := (S35Reed.In) ;
	Tracking11.Blocks[12] := NOT(S53Reed.In) ;
	Tracking11.ControlIN := Control.Achieved1 ;
	Tracking11.EMOStart := EMO.StartLatch ;
	Tracking11.ESClear := Control.ESClear ;
	Tracking11.BlockInhib := (Track922.Active) AND NOT((Tracking11.Blocks[6]) OR(Tracking11.Blocks[7])) ;
	Tracking11 ();
	Tracking11.ResMan := FALSE ;
	//RESET OF OUTPUTS
	Ax2.Active := FALSE ;
	Ax2.RaiseArms := FALSE ;
	Sol40Datum.Auto := FALSE ;
	CASE Tracking11.Index OF
		0: //RESET ALL TRACKBIT FOR SELECTED TRACKINGSECTION
			Track111 := TrackClear ;
			Track112 := TrackClear ;
			Track113 := TrackClear ;
			Track114 := TrackClear ;
			Track115 := TrackClear ;
		1: //TRACK FROM NOT Tracking10.Blocked (P) TO S32Reed.In (P)
			Track112 := TrackClear ;
			Track113 := TrackClear ;
			Track114 := TrackClear ;
			Track115 := TrackClear ;
			//FB INPUTS
			Track111.FixedIN := Tracking11.FixedOUT ;
			Track111.TimeoutEN := TRUE ;
			Track111.TimeoutACK := Warn.Ack ;
			Track111.TimeoutBlock := (Warn.Block) ;
			Track111.DelayPT := TrackDelayPT.PTTrack111 ;
			//FB CALL
			Track111 ();
			//FB OUTPUTS
			IF(Track111.Done) THEN
				Tracking11.IndexIN := 2 ;
			END_IF
		2: //TRACK FROM S32Reed.In (P) TO S6Photo.Int (P)
			Track111 := TrackClear ;
			Track113 := TrackClear ;
			Track114 := TrackClear ;
			Track115 := TrackClear ;
			//FB INPUTS
			Track112.FixedIN := Tracking11.FixedOUT ;
			Track112.Speed := Speeds.SpeedTrans ;
			Track112.TimeoutEN := TRUE ;
			Track112.TimeoutACK := Warn.Ack ;
			Track112.TimeoutBlock := (Warn.Block) ;
			Track112.DelayPT := TrackDelayPT.PTTrack112 ;
			//FB CALL
			Track112 ();
			//FB OUTPUTS
			CC2.o.Run[0] := Track112.RunOUT ;
			CC2.Inv.Scale1.x := Track112.SpeedOUT ;
			IF(Track112.Done) THEN
				Tracking11.IndexIN := 3 ;
			END_IF
		3: //TRACK FROM S6Photo.Int (P) TO S7Photo.Int (P)
			Track111 := TrackClear ;
			Track112 := TrackClear ;
			Track114 := TrackClear ;
			Track115 := TrackClear ;
			//FB INPUTS
			Track113.FixedIN := Tracking11.FixedOUT ;
			Track113.Speed := Speeds.SpeedSlow ;
			Track113.TimeoutEN := TRUE ;
			Track113.TimeoutACK := Warn.Ack ;
			Track113.TimeoutBlock := (Warn.Block) ;
			Track113.DelayPT := TrackDelayPT.PTTrack113 ;
			//FB CALL
			Track113 ();
			//FB OUTPUTS
			CC2.o.Run[0] := Track113.RunOUT ;
			CC2.Inv.Scale1.x := Track113.SpeedOUT ;
			IF(Track113.Done) THEN
				Tracking11.IndexIN := 4 ;
			END_IF
		4: //TRACK FROM S7Photo.Int (P) TO Ax2.SeekFin (P)
			Track111 := TrackClear ;
			Track112 := TrackClear ;
			Track113 := TrackClear ;
			Track115 := TrackClear ;
			//FB INPUTS
			Track114.FixedIN := Tracking11.FixedOUT ;
			//FB CALL
			Track114 ();
			//FB OUTPUTS
			IF NOT(Ax2.HiVol) THEN
				Ax2.Seek1 := (Track114.SolOUT) AND NOT(Ax2.Block) ;
			ELSE
				Tracking11.IndexIN := 5 ;
			END_IF
			IF(Track114.Done) THEN
				Tracking11.IndexIN := 5 ;
			END_IF
		5: //TRACK FROM Ax2.SeekFin (P) TO NOT Tracking11.Blocked (-)
			Track111 := TrackClear ;
			Track112 := TrackClear ;
			Track113 := TrackClear ;
			Track114 := TrackClear ;
			//FB INPUTS
			Track115.FixedIN := Tracking11.FixedOUT ;
			//FB CALL
			Track115 ();
			//FB OUTPUTS
			Sol40Datum.Auto := (Track115.SolOUT) ;
			Ax2.RaiseArms := (Track115.SolOUT) ;
			IF(Track115.Done) THEN
				Tracking11.IndexIN := 0 ;
				Tracking20.IndexIN := 1 ;
				Tracking94.IndexIN := 1 ;
				Tracking20.LengthIN := Tracking11.Length ;
				Tracking20.RowBlockIN := Tracking11.RowBlock;
			END_IF
	END_CASE

	//TRACKBIT DONE CONDITIONS
	Track111.DoneIN := EDGEPOS(S32Reed.In) ;
	Track112.DoneIN := EDGEPOS(S6Photo.Int) ;
	Track113.DoneIN := EDGEPOS(S7Photo.Int) ;
	Track114.DoneIN := EDGEPOS(Ax2.SeekFin) ;
	Track115.DoneIN := NOT(Tracking11.Blocked) ;

	Ax2.Active := Track114.Active ;

	//TRACKINGSECTION END BLOCK CONDITIONS
	Tracking94.ControlIN := Control.Achieved1 ;
	Tracking94.EMOStart := EMO.StartLatch ;
	Tracking94.ESClear := Control.ESClear ;
	Tracking94 ();
	Tracking94.ResMan := FALSE ;
	CASE Tracking94.Index OF
		0: //RESET ALL TRACKBIT FOR SELECTED TRACKINGSECTION
			Track941 := TrackClear ;
		1: //TRACK FROM NOT Tracking11.Blocked (-) TO S7Photo.Int (N)
			//FB INPUTS
			Track941.FixedIN := Tracking94.FixedOUT ;
			Track941.RunBlock := (Track201.TimeoutOUT) OR(Track204.TimeoutOUT) OR NOT((Track201.RunOUT) OR(Track204.RunOUT)) ;
			IF (ProcessMode.In) THEN
				Track941.Speed := Speeds.SpeedSeamSlow;
			ELSE
				Track941.Speed := Speeds.SpeedSeam ;
			END_IF
			//FB CALL
			Track941 ();
			//FB OUTPUTS
			CC2.o.Run[0] := Track941.RunOUT ;
			CC2.Inv.Scale1.x := Track941.SpeedOUT ;
			IF(Track941.Done) THEN
				Tracking94.IndexIN := 0 ;
			END_IF
	END_CASE

	//TRACKBIT DONE CONDITIONS
	Track941.DoneIN := EDGENEG(S7Photo.Int) ;

	//MANUAL RESET CONDITIONS FOR CONCURRENT TRACKBIT
	Tracking94.ResMan := Tracking20.ResMan ;
	IF(Tracking20.IndexIN = 0) THEN
		Tracking94.IndexIN := 0 ;
	END_IF

END_PROGRAM
```

### Program Logical/Automatic/ConSeam2 (IEC) - Seaming 2 conveyor

#### ConSeam2Cyclic.st - Cyclic code
```iecst
(********************************************************************
 * COPYRIGHT --
 ********************************************************************
 * Program: ConSeam2
 * File: ConSeam2Cyclic.st
 * Author: nicke
 ********************************************************************
 * Implementation of program ConSeam2
 ********************************************************************)

PROGRAM _CYCLIC

   //TRACKINGSECTION END BLOCK CONDITIONS
	Tracking20.Blocks[0] := (Tracking30.Busy) ;
	Tracking20.Blocks[2] := (CB1.Input.Fault) ;
	Tracking20.Blocks[9] := (S14Photo.Int) ;
	Tracking20.Blocks[10] := (S15Photo.Int) ;
	Tracking20.ControlIN := Control.Achieved1 ;
	Tracking20.EMOStart := EMO.StartLatch ;
	Tracking20.ESClear := Control.ESClear ;
	Tracking20.BlockInhib := (Track401.Active) ;
	Tracking20 ();
	Tracking20.ResMan := FALSE ;
	//RESET OF OUTPUTS
	Seaming.Start2 := FALSE ;
	Seaming.Stop2 := FALSE ;
	Sol32Pal3.Auto := FALSE ;
	CASE Tracking20.Index OF
		0: //RESET ALL TRACKBIT FOR SELECTED TRACKINGSECTION
			Track201 := TrackClear ;
			Track202 := TrackClear ;
			Track203 := TrackClear ;
			Track204 := TrackClear ;
			Track205 := TrackClear ;
			Track206 := TrackClear ;
			Track207 := TrackClear ;
			Track208 := TrackClear ;
		1: //TRACK FROM NOT Tracking11.Blocked (-) TO S12Photo.Int (P)
			Track202 := TrackClear ;
			Track203 := TrackClear ;
			Track204 := TrackClear ;
			Track205 := TrackClear ;
			Track206 := TrackClear ;
			Track207 := TrackClear ;
			Track208 := TrackClear ;
			//FB INPUTS
			Track201.FixedIN := Tracking20.FixedOUT ;
			IF (ProcessMode.In) THEN
				Track201.Speed := Speeds.SpeedSeamSlow;
			ELSE
				Track201.Speed := Speeds.SpeedSeam ;
			END_IF
			Track201.RunBlock := NOT(SeamersII.DoneOUT[2]) ;
			Track201.TimeoutEN := TRUE ;
			Track201.TimeoutACK := Warn.Ack ;
			Track201.TimeoutBlock := (Warn.Block) ;
			Track201.DelayPT := TrackDelayPT.PTTrack201 ;
			//FB CALL
			Track201 ();
			//FB OUTPUTS
			CS2.o.Run[0] := Track201.RunOUT ;
			CV2.o.Run[0] := Track201.RunOUT ;
			CC3.o.Run[0] := Track201.RunOUT ;
			CS2.Inv.Scale1.x := Track201.SpeedOUT ;
			CV2.Inv.Scale1.x := Track201.SpeedOUT ;
			CC3.Inv.Scale1.x := Track201.SpeedOUT ;
			Sol40Datum.Auto := (Track201.SolOUT) AND(Tracking94.Busy) ;
			Ax2.RaiseArms := (Track201.SolOUT) ;
			IF(Track201.Done) THEN
				Tracking20.IndexIN := 4 ;
				Tracking20.WidthIN := Ax2.Measure/10.0 ;
			END_IF
		2: //TRACK FROM S8Photo.Int (P) TO S8Photo.Int (N)
			Track201 := TrackClear ;
			Track203 := TrackClear ;
			Track204 := TrackClear ;
			Track205 := TrackClear ;
			Track206 := TrackClear ;
			Track207 := TrackClear ;
			Track208 := TrackClear ;
			//FB INPUTS
//			Track202.FixedIN := Tracking20.FixedOUT ;
//			IF (ProcessMode.In) THEN
//				Track202.Speed := Speeds.SpeedSeamSlow;
//			ELSE
//				Track202.Speed := Speeds.SpeedSeam ;
//			END_IF
//			Track202.RunBlock := NOT(SeamersII.DoneOUT[2]) ;
//			Track202.TimeoutEN := TRUE ;
//			Track202.TimeoutACK := Warn.Ack ;
//			Track202.TimeoutBlock := (Warn.Block) ;
//			Track202.DelayPT := TrackDelayPT.PTTrack202 ;
//			//FB CALL
//			Track202 ();
//			//FB OUTPUTS
//			CS2.o.Run[0] := Track202.RunOUT ;
//			CV2.o.Run[0] := Track202.RunOUT ;
//			CC3.o.Run[0] := Track202.RunOUT ;
//			CS2.Inv.Scale1.x := Track202.SpeedOUT ;
//			CV2.Inv.Scale1.x := Track202.SpeedOUT ;
//			CC3.Inv.Scale1.x := Track202.SpeedOUT ;
//			Sol40Datum.Auto := (Track202.SolOUT) AND(Tracking94.Busy) ;
//			Seaming.Start2 := (Track202.SolOUT) ;
//			Ax2.RaiseArms := (Track202.SolOUT) ;
//			IF(Track202.Done) THEN
//				Tracking20.IndexIN := 4 ;
//			END_IF
		3: //TRACK FROM S8Photo.Int (N) TO Belts2.Done (P)
			Track201 := TrackClear ;
			Track202 := TrackClear ;
			Track204 := TrackClear ;
			Track205 := TrackClear ;
			Track206 := TrackClear ;
			Track207 := TrackClear ;
			Track208 := TrackClear ;
			//FB INPUTS
//			Track203.FixedIN := Tracking20.FixedOUT ;
//			IF (ProcessMode.In) THEN
//				Track203.Speed := Speeds.SpeedSeamSlow;
//			ELSE
//				Track203.Speed := Speeds.SpeedSeam ;
//			END_IF
//			Track203.RunBlock := NOT(SeamersII.DoneOUT[2]) ;
//			//FB CALL
//			Track203 ();
//			//FB OUTPUTS
//			CS2.o.Run[0] := Track203.RunOUT ;
//			CV2.o.Run[0] := Track203.RunOUT ;
//			CC3.o.Run[0] := Track203.RunOUT ;
//			CS2.Inv.Scale1.x := Track203.SpeedOUT ;
//			CV2.Inv.Scale1.x := Track203.SpeedOUT ;
//			CC3.Inv.Scale1.x := Track203.SpeedOUT ;
//			Seaming.Stop2 := (Track203.SolOUT) ;
//			Ax2.RaiseArms := (Track203.SolOUT) ;
//			IF(Track203.Done) THEN
//				Tracking20.IndexIN := 4 ;
//				Tracking20.WidthIN := Ax2.Measure/10.0 ;
//			END_IF
		4: //TRACK FROM S12Photo.Int (P) TO S12Photo.Int (N)
			Track201 := TrackClear ;
			Track202 := TrackClear ;
			Track203 := TrackClear ;
			Track205 := TrackClear ;
			Track206 := TrackClear ;
			Track207 := TrackClear ;
			Track208 := TrackClear ;
			//FB INPUTS
			Track204.FixedIN := Tracking20.FixedOUT ;
			IF (ProcessMode.In) THEN
				Track204.Speed := Speeds.SpeedSeamSlow;
				Track204.DelayPT := REAL_TO_UDINT((UDINT_TO_REAL(TrackDelayPT.PTTrack204)) * (Speeds.SpeedSeam/Speeds.SpeedSeamSlow)) ;
			ELSE
				Track204.Speed := Speeds.SpeedSeam ;
				Track204.DelayPT := TrackDelayPT.PTTrack204 ;
			END_IF
			Track204.TimeoutEN := TRUE ;
			Track204.TimeoutACK := Warn.Ack ;
			Track204.TimeoutBlock := (Warn.Block) ;
			//FB CALL
			Track204 ();
			//FB OUTPUTS
			CS2.o.Run[0] := Track204.RunOUT ;
			CV2.o.Run[0] := Track204.RunOUT ;
			CC3.o.Run[0] := Track204.RunOUT ;
			CS2.Inv.Scale1.x := Track204.SpeedOUT ;
			CV2.Inv.Scale1.x := Track204.SpeedOUT ;
			CC3.Inv.Scale1.x := Track204.SpeedOUT ;
			Ax2.RaiseArms := (Track204.SolOUT) ;
			IF(Track204.Done) THEN
				Tracking20.IndexIN := 5 ;
			END_IF
		5: //TRACK FROM S12Photo.Int (N) TO Track205.DelayTON.Q (P)
			Track201 := TrackClear ;
			Track202 := TrackClear ;
			Track203 := TrackClear ;
			Track204 := TrackClear ;
			Track206 := TrackClear ;
			Track207 := TrackClear ;
			Track208 := TrackClear ;
			//FB INPUTS
			Track205.FixedIN := Tracking20.FixedOUT ;
			Track205.Speed := Speeds.SpeedSlow ;
			Track205.TrackDelayEN := TRUE ;
			Track205.DelayPT := TrackDelayPT.PTTrack205 ;
			//FB CALL
			Track205 ();
			//FB OUTPUTS
			CC3.o.Run[0] := Track205.RunOUT ;
			CC3.Inv.Scale1.x := Track205.SpeedOUT ;
			IF(Track205.Done) THEN
				Tracking20.IndexIN := 6 ;
			END_IF
		6: //TRACK FROM Track205.DelayTON.Q (P) TO Track206.DelayTON.Q (P)
			Track201 := TrackClear ;
			Track202 := TrackClear ;
			Track203 := TrackClear ;
			Track204 := TrackClear ;
			Track205 := TrackClear ;
			Track207 := TrackClear ;
			Track208 := TrackClear ;
			//FB INPUTS
			Track206.FixedIN := Tracking20.FixedOUT ;
			Track206.Speed := Speeds.SpeedSlow ;
			Track206.TrackDelayEN := TRUE ;
			Track206.DelayPT := TrackDelayPT.PTTrack206 ;
			//FB CALL
			Track206 ();
			//FB OUTPUTS
			CC3.o.Rev[0] := Track206.RunOUT ;
			CC3.Inv.Scale1.x := Track206.SpeedOUT ;
			IF(Track206.Done) THEN
				Tracking20.IndexIN := 7 ;
			END_IF
		7: //TRACK FROM Track206.DelayTON.Q (P) TO S35Reed.In (P)
			Track201 := TrackClear ;
			Track202 := TrackClear ;
			Track203 := TrackClear ;
			Track204 := TrackClear ;
			Track205 := TrackClear ;
			Track206 := TrackClear ;
			Track208 := TrackClear ;
			//FB INPUTS
			Track207.FixedIN := Tracking20.FixedOUT ;
			Track207.TimeoutEN := TRUE ;
			Track207.TimeoutACK := Warn.Ack ;
			Track207.TimeoutBlock := (Warn.Block) ;
			Track207.DelayPT := TrackDelayPT.PTTrack207 ;
			//FB CALL
			Track207 ();
			//FB OUTPUTS
			Sol32Pal3.Auto := (Track207.SolOUT) ;
			IF(Track207.Done) THEN
				Tracking20.IndexIN := 8 ;
			END_IF
		8: //TRACK FROM S35Reed.In (P) TO NOT Tracking20.Blocked (-)
			Track201 := TrackClear ;
			Track202 := TrackClear ;
			Track203 := TrackClear ;
			Track204 := TrackClear ;
			Track205 := TrackClear ;
			Track206 := TrackClear ;
			Track207 := TrackClear ;
			//FB INPUTS
			Track208.FixedIN := Tracking20.FixedOUT ;
			//FB CALL
			Track208 ();
			//FB OUTPUTS
			Sol32Pal3.Auto := (Track208.SolOUT) ;
			IF(Track208.Done) THEN
				Tracking20.IndexIN := 0 ;
				Tracking30.IndexIN := 1 ;
				Tracking92.IndexIN := 1 ;
				Tracking30.LengthIN := Tracking20.Length ;
				Tracking30.WidthIN := Tracking20.Width ;
				Tracking30.RowBlockIN := Tracking20.RowBlock ;
			END_IF
	END_CASE

	//TRACKBIT DONE CONDITIONS
	Track201.DoneIN := EDGEPOS(S12Photo.Int) ;
//	Track202.DoneIN := EDGENEG(S8Photo.Int) ;
//	Track203.DoneIN := EDGEPOS(Belts2.Done) ;
	Track204.DoneIN := EDGENEG(S12Photo.Int) ;
	Track207.DoneIN := EDGEPOS(S35Reed.In) ;
	Track208.DoneIN := NOT(Tracking20.Blocked) ;

	//TRACKINGSECTION END BLOCK CONDITIONS
	Tracking92.ControlIN := Control.Achieved1 ;
	Tracking92.EMOStart := EMO.StartLatch ;
	Tracking92.ESClear := Control.ESClear ;
	Tracking92 ();
	Tracking92.ResMan := FALSE ;
	CASE Tracking92.Index OF
		0: //RESET ALL TRACKBIT FOR SELECTED TRACKINGSECTION
			Track921 := TrackClear ;
			Track922 := TrackClear ;
		1: //TRACK FROM NOT Tracking20.Blocked (-) TO Track921.DelayTON.Q (P)
			Track922 := TrackClear ;
			//FB INPUTS
			Track921.FixedIN := Tracking92.FixedOUT ;
			Track921.RunBlock := (Track301.TimeoutOUT) OR(Track302.TimeoutOUT) ;
			Track921.Speed := Speeds.SpeedExit ;
			Track921.TrackDelayEN := TRUE ;
			Track921.DelayPT := TrackDelayPT.PTTrack921 ;
			//FB CALL
			Track921 ();
			//FB OUTPUTS
			CC4.o.Run[0] := Track921.RunOUT ;
			CC4.Inv.Scale1.x := Track921.SpeedOUT ;
			Sol32Pal3.Auto := (Track921.SolOUT) ;
			IF(Track921.Done) THEN
				Tracking92.IndexIN := 2 ;
			END_IF
		2: //TRACK FROM Track521.DelayTON.Q (P) TO  NOT S13Photo.Int (-)
			Track921 := TrackClear ;
			//FB INPUTS
			Track922.FixedIN := Tracking92.FixedOUT ;
			Track922.RunBlock := (Track301.TimeoutOUT) OR(Track302.TimeoutOUT) OR((Track302.Active)AND(Tracking30.Blocked)) ;
			Track922.Speed := Speeds.SpeedExit ;
			//FB CALL
			Track922 ();
			//FB OUTPUTS
			CC4.o.Run[0] := Track922.RunOUT ;
			CC4.Inv.Scale1.x := Track922.SpeedOUT ;
			Sol32Pal3.Auto := (Track922.SolOUT) ;
			IF(Track922.Done) THEN
				Tracking92.IndexIN := 0 ;
			END_IF
	END_CASE

	//TRACKBIT DONE CONDITIONS
	Track922.DoneIN := NOT(S13Photo.Int) ;

	//MANUAL RESET CONDITIONS FOR CONCURRENT TRACKBIT
	Tracking92.ResMan := Tracking30.ResMan ;
	IF(Tracking30.IndexIN = 0) THEN
		Tracking92.IndexIN := 0 ;
	END_IF

END_PROGRAM
```

### Program Logical/Automatic/ConBuffers (IEC) - Buffer conveyors
